  MoveL 8069 to (229.18, 36.07, 116.27) mm, rotated rx -180 ry 0 rz 180 deg; joints [-27.539, 54.39, -86.932, 31.738, 118.488, 16.437]
  MoveL 8070 to (229.18, 36.07, 116.27) mm, rotated rx -180 ry 0 rz 180 deg; joints [-27.539, 54.39, -86.932, 31.738, 118.488, 16.437]
  Call Extruder(197.85836)
  MoveL 8071 to (229.38, 36.12, 116.27) mm, rotated rx 180 ry 0 rz 180 deg; joints [-27.499, 54.413, -86.932, 31.688, 118.48, 16.403]
  MoveL 8072 to (229.38, 36.12, 116.27) mm, rotated rx 180 ry 0 rz 180 deg; joints [-27.499, 54.413, -86.932, 31.688, 118.48, 16.403]
  Call Extruder(197.97344)
  MoveL 8073 to (229.59, 36.16, 116.27) mm, rotated rx -180 ry 0 rz 180 deg; joints [-27.458, 54.436, -86.932, 31.638, 118.472, 16.368]
  MoveL 8074 to (229.59, 36.16, 116.27) mm, rotated rx -180 ry 0 rz 180 deg; joints [-27.458, 54.436, -86.932, 31.638, 118.472, 16.368]
  Call Extruder(198.09430)
  MoveL 8075 to (229.8, 36.21, 116.27) mm, rotated rx -180 ry 0 rz -180 deg; joints [-27.422, 54.459, -86.932, 31.591, 118.461, 16.335]
  MoveL 8076 to (229.8, 36.21, 116.27) mm, rotated rx -180 ry 0 rz -180 deg; joints [-27.422, 54.459, -86.932, 31.591, 118.461, 16.335]
  Call Extruder(198.22115)
  MoveL 8077 to (230.02, 36.28, 116.27) mm, rotated rx -180 ry 0 rz 180 deg; joints [-27.39, 54.485, -86.931, 31.549, 118.448, 16.303]
  MoveL 8078 to (230.02, 36.28, 116.27) mm, rotated rx -180 ry 0 rz 180 deg; joints [-27.39, 54.485, -86.931, 31.549, 118.448, 16.303]
  Call Extruder(198.33995)
  MoveL 8079 to (230.22, 36.34, 116.27) mm, rotated rx -180 ry 0 rz 180 deg; joints [-27.361, 54.508, -86.931, 31.51, 118.436, 16.274]
  MoveL 8080 to (230.22, 36.34, 116.27) mm, rotated rx -180 ry 0 rz 180 deg; joints [-27.361, 54.508, -86.931, 31.51, 118.436, 16.274]
  Call Extruder(198.45066)
  MoveL 8081 to (230.41, 36.4, 116.27) mm, rotated rx -180 ry 0 rz 180 deg; joints [-27.336, 54.53, -86.931, 31.477, 118.424, 16.248]
  MoveL 8082 to (230.41, 36.4, 116.27) mm, rotated rx -180 ry 0 rz 180 deg; joints [-27.336, 54.53, -86.931, 31.477, 118.424, 16.248]
  Call Extruder(198.56179)
  MoveL 8083 to (230.6, 36.46, 116.27) mm, rotated rx -180 ry 0 rz 180 deg; joints [-27.311, 54.552, -86.93, 31.444, 118.412, 16.222]
  MoveL 8084 to (230.6, 36.46, 116.27) mm, rotated rx -180 ry 0 rz 180 deg; joints [-27.311, 54.552, -86.93, 31.444, 118.412, 16.222]
  Call Extruder(198.67341)
  MoveL 8085 to (230.79, 36.52, 116.27) mm, rotated rx -180 ry 0 rz 180 deg; joints [-27.288, 54.574, -86.93, 31.412, 118.4, 16.196]
  MoveL 8086 to (230.79, 36.52, 116.27) mm, rotated rx -180 ry 0 rz 180 deg; joints [-27.288, 54.574, -86.93, 31.412, 118.4, 16.196]
  Call Extruder(198.78553)
  MoveL 8087 to (230.98, 36.58, 116.27) mm, rotated rx 180 ry 0 rz 180 deg; joints [-27.265, 54.596, -86.93, 31.381, 118.387, 16.171]
  MoveL 8088 to (230.98, 36.58, 116.27) mm, rotated rx 180 ry 0 rz 180 deg; joints [-27.265, 54.596, -86.93, 31.381, 118.387, 16.171]
  Call Extruder(198.89810)
  MoveL 8089 to (231.17, 36.64, 116.27) mm, rotated rx 180 ry 0 rz 180 deg; joints [-27.242, 54.618, -86.929, 31.349, 118.374, 16.146]
  MoveL 8090 to (231.17, 36.64, 116.27) mm, rotated rx 180 ry 0 rz 180 deg; joints [-27.242, 54.618, -86.929, 31.349, 118.374, 16.146]
  Call Extruder(199.01111)
  MoveL 8091 to (231.35, 36.7, 116.27) mm, rotated rx 180 ry 0 rz 180 deg; joints [-27.219, 54.64, -86.929, 31.318, 118.362, 16.121]
  MoveL 8092 to (231.35, 36.7, 116.27) mm, rotated rx 180 ry 0 rz 180 deg; joints [-27.219, 54.64, -86.929, 31.318, 118.362, 16.121]
  Call Extruder(199.12456)
  MoveL 8093 to (231.54, 36.76, 116.27) mm, rotated rx 180 ry 0 rz 180 deg; joints [-27.197, 54.662, -86.928, 31.287, 118.349, 16.096]
  MoveL 8094 to (231.54, 36.76, 116.27) mm, rotated rx 180 ry 0 rz 180 deg; joints [-27.197, 54.662, -86.928, 31.287, 118.349, 16.096]
  Call Extruder(199.27220)
  MoveL 8095 to (231.78, 36.85, 116.27) mm, rotated rx -180 ry 0 rz -180 deg; joints [-27.176, 54.691, -86.928, 31.257, 118.329, 16.068]
  MoveL 8096 to (231.78, 36.85, 116.27) mm, rotated rx -180 ry 0 rz -180 deg; joints [-27.176, 54.691, -86.928, 31.257, 118.329, 16.068]
  Call Extruder(199.45454)
  MoveL 8097 to (232.07, 36.97, 116.27) mm, rotated rx -180 ry 0 rz 180 deg; joints [-27.158, 54.726, -86.927, 31.227, 118.304, 16.038]
  MoveL 8098 to (232.07, 36.97, 116.27) mm, rotated rx -180 ry 0 rz 180 deg; joints [-27.158, 54.726, -86.927, 31.227, 118.304, 16.038]
  Call Extruder(199.63764)
  MoveL 8099 to (232.37, 37.1, 116.27) mm, rotated rx 180 ry 0 rz 180 deg; joints [-27.139, 54.761, -86.926, 31.196, 118.278, 16.007]
  MoveL 8100 to (232.37, 37.1, 116.27) mm, rotated rx 180 ry 0 rz 180 deg; joints [-27.139, 54.761, -86.926, 31.196, 118.278, 16.007]
  Call Extruder(199.79534)
  MoveL 8101 to (232.62, 37.2, 116.27) mm, rotated rx 180 ry 0 rz 180 deg; joints [-27.127, 54.791, -86.926, 31.174, 118.255, 15.982]
  MoveL 8102 to (232.62, 37.2, 116.27) mm, rotated rx 180 ry 0 rz 180 deg; joints [-27.127, 54.791, -86.926, 31.174, 118.255, 15.982]
  Call Extruder(199.95364)
  MoveL 8103 to (232.87, 37.31, 116.27) mm, rotated rx -180 ry 0 rz -180 deg; joints [-27.114, 54.822, -86.925, 31.151, 118.232, 15.957]
  MoveL 8104 to (232.87, 37.31, 116.27) mm, rotated rx -180 ry 0 rz -180 deg; joints [-27.114, 54.822, -86.925, 31.151, 118.232, 15.957]
  Call Extruder(200.13566)
  MoveL 8105 to (233.14, 37.45, 116.27) mm, rotated rx -180 ry 0 rz 180 deg; joints [-27.114, 54.856, -86.924, 31.141, 118.202, 15.936]
  MoveL 8106 to (233.14, 37.45, 116.27) mm, rotated rx -180 ry 0 rz 180 deg; joints [-27.114, 54.856, -86.924, 31.141, 118.202, 15.936]
  Call Extruder(200.34222)
  MoveL 8107 to (233.45, 37.63, 116.27) mm, rotated rx 180 ry 0 rz 180 deg; joints [-27.126, 54.895, -86.923, 31.143, 118.164, 15.919]
  MoveL 8108 to (233.45, 37.63, 116.27) mm, rotated rx 180 ry 0 rz 180 deg; joints [-27.126, 54.895, -86.923, 31.143, 118.164, 15.919]
  Call Extruder(200.54955)
  MoveL 8109 to (233.75, 37.8, 116.27) mm, rotated rx -180 ry 0 rz 180 deg; joints [-27.138, 54.935, -86.922, 31.145, 118.126, 15.901]
  MoveL 8110 to (233.75, 37.8, 116.27) mm, rotated rx -180 ry 0 rz 180 deg; joints [-27.138, 54.935, -86.922, 31.145, 118.126, 15.901]
  Call Extruder(200.75767)
  MoveL 8111 to (234.05, 37.98, 116.27) mm, rotated rx 180 ry 0 rz -180 deg; joints [-27.15, 54.974, -86.921, 31.148, 118.089, 15.884]
  MoveL 8112 to (234.05, 37.98, 116.27) mm, rotated rx 180 ry 0 rz -180 deg; joints [-27.15, 54.974, -86.921, 31.148, 118.089, 15.884]
  Call Extruder(200.87539)
  MoveL 8113 to (234.23, 38.08, 116.27) mm, rotated rx 180 ry 0 rz 180 deg; joints [-27.157, 54.996, -86.921, 31.149, 118.067, 15.875]
  MoveL 8114 to (234.23, 38.08, 116.27) mm, rotated rx 180 ry 0 rz 180 deg; joints [-27.157, 54.996, -86.921, 31.149, 118.067, 15.875]
  Call Extruder(201.20821)
  MoveL 8115 to (234.68, 38.4, 116.27) mm, rotated rx -180 ry 0 rz 180 deg; joints [-27.216, 55.057, -86.919, 31.196, 117.997, 15.868]
  MoveL 8116 to (234.68, 38.4, 116.27) mm, rotated rx -180 ry 0 rz 180 deg; joints [-27.216, 55.057, -86.919, 31.196, 117.997, 15.868]
  Call Extruder(201.54222)
  MoveL 8117 to (235.13, 38.73, 116.27) mm, rotated rx -180 ry 0 rz 180 deg; joints [-27.274, 55.119, -86.917, 31.241, 117.927, 15.86]
  MoveL 8118 to (235.13, 38.73, 116.27) mm, rotated rx -180 ry 0 rz 180 deg; joints [-27.274, 55.119, -86.917, 31.241, 117.927, 15.86]
  Call Extruder(201.70980)
  MoveL 8119 to (235.35, 38.9, 116.27) mm, rotated rx -180 ry 0 rz 180 deg; joints [-27.302, 55.149, -86.916, 31.264, 117.892, 15.856]
  Call Extruder(202.53913)
  MoveL 8120 to (236.39, 39.81, 116.27) mm, rotated rx 180 ry 0 rz 180 deg; joints [-27.525, 55.298, -86.91, 31.463, 117.7, 15.878]
  Call Extruder(203.17020)
  MoveL 8121 to (237.09, 40.59, 116.27) mm, rotated rx -180 ry 0 rz -180 deg; joints [-27.771, 55.407, -86.906, 31.7, 117.536, 15.935]
  MoveL 8122 to (237.09, 40.59, 116.27) mm, rotated rx -180 ry 0 rz -180 deg; joints [-27.771, 55.407, -86.906, 31.7, 117.536, 15.935]
  Call Extruder(203.36780)
  MoveL 8123 to (237.3, 40.85, 116.27) mm, rotated rx 180 ry 0 rz 180 deg; joints [-27.851, 55.441, -86.905, 31.777, 117.484, 15.954]
  Call Extruder(203.70181)
  MoveL 8124 to (237.63, 41.3, 116.27) mm, rotated rx 180 ry 0 rz 180 deg; joints [-28.012, 55.496, -86.902, 31.935, 117.39, 16]
  MoveL 8125 to (237.63, 41.3, 116.27) mm, rotated rx 180 ry 0 rz 180 deg; joints [-28.012, 55.496, -86.902, 31.935, 117.39, 16]
  Call Extruder(204.03463)
  MoveL 8126 to (237.96, 41.75, 116.27) mm, rotated rx 180 ry 0 rz 180 deg; joints [-28.17, 55.551, -86.9, 32.09, 117.298, 16.044]
  MoveL 8127 to (237.96, 41.75, 116.27) mm, rotated rx 180 ry 0 rz 180 deg; joints [-28.17, 55.551, -86.9, 32.09, 117.298, 16.044]
  Call Extruder(204.21387)
  MoveL 8128 to (238.13, 41.99, 116.27) mm, rotated rx 180 ry 0 rz 180 deg; joints [-28.256, 55.581, -86.898, 32.174, 117.247, 16.068]
  MoveL 8129 to (238.13, 41.99, 116.27) mm, rotated rx 180 ry 0 rz 180 deg; joints [-28.256, 55.581, -86.898, 32.174, 117.247, 16.068]
  Call Extruder(204.42198)
  MoveL 8130 to (238.31, 42.3, 116.27) mm, rotated rx -180 ry 0 rz 180 deg; joints [-28.375, 55.614, -86.897, 32.293, 117.185, 16.106]
  MoveL 8131 to (238.31, 42.3, 116.27) mm, rotated rx -180 ry 0 rz 180 deg; joints [-28.375, 55.614, -86.897, 32.293, 117.185, 16.106]
  Call Extruder(204.62931)
  MoveL 8132 to (238.49, 42.6, 116.27) mm, rotated rx -180 ry 0 rz -180 deg; joints [-28.493, 55.647, -86.895, 32.412, 117.123, 16.143]
  MoveL 8133 to (238.49, 42.6, 116.27) mm, rotated rx -180 ry 0 rz -180 deg; joints [-28.493, 55.647, -86.895, 32.412, 117.123, 16.143]
  Call Extruder(204.83587)
  MoveL 8134 to (238.66, 42.91, 116.27) mm, rotated rx -180 ry 0 rz -180 deg; joints [-28.61, 55.68, -86.893, 32.528, 117.061, 16.18]
  MoveL 8135 to (238.66, 42.91, 116.27) mm, rotated rx -180 ry 0 rz -180 deg; joints [-28.61, 55.68, -86.893, 32.528, 117.061, 16.18]
  Call Extruder(205.04165)
  MoveL 8136 to (238.84, 43.21, 116.27) mm, rotated rx -180 ry 0 rz 180 deg; joints [-28.727, 55.713, -86.892, 32.645, 117, 16.216]
  MoveL 8137 to (238.84, 43.21, 116.27) mm, rotated rx -180 ry 0 rz 180 deg; joints [-28.727, 55.713, -86.892, 32.645, 117, 16.216]
  Call Extruder(205.19996)
  MoveL 8138 to (238.94, 43.46, 116.27) mm, rotated rx -180 ry 0 rz 180 deg; joints [-28.834, 55.737, -86.89, 32.753, 116.949, 16.253]
  MoveL 8139 to (238.94, 43.46, 116.27) mm, rotated rx -180 ry 0 rz 180 deg; joints [-28.834, 55.737, -86.89, 32.753, 116.949, 16.253]
  Call Extruder(205.35767)
  MoveL 8140 to (239.05, 43.71, 116.27) mm, rotated rx 180 ry 0 rz 180 deg; joints [-28.939, 55.76, -86.889, 32.86, 116.899, 16.29]
  MoveL 8141 to (239.05, 43.71, 116.27) mm, rotated rx 180 ry 0 rz 180 deg; joints [-28.939, 55.76, -86.889, 32.86, 116.899, 16.29]
  Call Extruder(205.52776)
  MoveL 8142 to (239.17, 43.98, 116.27) mm, rotated rx 180 ry 0 rz 180 deg; joints [-29.054, 55.785, -86.888, 32.976, 116.844, 16.329]
  MoveL 8143 to (239.17, 43.98, 116.27) mm, rotated rx 180 ry 0 rz 180 deg; joints [-29.054, 55.785, -86.888, 32.976, 116.844, 16.329]
  Call Extruder(205.71010)
  MoveL 8144 to (239.29, 44.27, 116.27) mm, rotated rx -180 ry 0 rz 180 deg; joints [-29.178, 55.813, -86.886, 33.101, 116.785, 16.372]
  MoveL 8145 to (239.29, 44.27, 116.27) mm, rotated rx -180 ry 0 rz 180 deg; joints [-29.178, 55.813, -86.886, 33.101, 116.785, 16.372]
  Call Extruder(205.89168)
  MoveL 8146 to (239.41, 44.56, 116.27) mm, rotated rx 180 ry 0 rz -180 deg; joints [-29.301, 55.84, -86.885, 33.226, 116.726, 16.414]
  MoveL 8147 to (239.41, 44.56, 116.27) mm, rotated rx 180 ry 0 rz -180 deg; joints [-29.301, 55.84, -86.885, 33.226, 116.726, 16.414]
  Call Extruder(206.00513)
  MoveL 8148 to (239.47, 44.75, 116.27) mm, rotated rx -180 ry 0 rz 180 deg; joints [-29.385, 55.856, -86.884, 33.311, 116.688, 16.444]
  MoveL 8149 to (239.47, 44.75, 116.27) mm, rotated rx -180 ry 0 rz 180 deg; joints [-29.385, 55.856, -86.884, 33.311, 116.688, 16.444]
  Call Extruder(206.11815)
  MoveL 8150 to (239.53, 44.94, 116.27) mm, rotated rx 180 ry 0 rz -180 deg; joints [-29.47, 55.872, -86.883, 33.397, 116.65, 16.475]
  MoveL 8151 to (239.53, 44.94, 116.27) mm, rotated rx 180 ry 0 rz -180 deg; joints [-29.47, 55.872, -86.883, 33.397, 116.65, 16.475]
  Call Extruder(206.23072)
  MoveL 8152 to (239.59, 45.13, 116.27) mm, rotated rx -180 ry 0 rz 180 deg; joints [-29.553, 55.888, -86.882, 33.482, 116.612, 16.504]
  MoveL 8153 to (239.59, 45.13, 116.27) mm, rotated rx -180 ry 0 rz 180 deg; joints [-29.553, 55.888, -86.882, 33.482, 116.612, 16.504]
  Call Extruder(206.34284)
  MoveL 8154 to (239.65, 45.32, 116.27) mm, rotated rx 180 ry 0 rz -180 deg; joints [-29.637, 55.904, -86.881, 33.568, 116.574, 16.534]
  MoveL 8155 to (239.65, 45.32, 116.27) mm, rotated rx 180 ry 0 rz -180 deg; joints [-29.637, 55.904, -86.881, 33.568, 116.574, 16.534]
  Call Extruder(206.45452)
  MoveL 8156 to (239.71, 45.51, 116.27) mm, rotated rx 180 ry 0 rz 180 deg; joints [-29.72, 55.92, -86.88, 33.652, 116.537, 16.563]
  MoveL 8157 to (239.71, 45.51, 116.27) mm, rotated rx 180 ry 0 rz 180 deg; joints [-29.72, 55.92, -86.88, 33.652, 116.537, 16.563]
  Call Extruder(206.58559)
  MoveL 8158 to (239.78, 45.73, 116.27) mm, rotated rx -180 ry 0 rz 180 deg; joints [-29.821, 55.939, -86.879, 33.754, 116.492, 16.599]
  MoveL 8159 to (239.78, 45.73, 116.27) mm, rotated rx -180 ry 0 rz 180 deg; joints [-29.821, 55.939, -86.879, 33.754, 116.492, 16.599]
  Call Extruder(206.71610)
  MoveL 8160 to (239.85, 45.95, 116.27) mm, rotated rx 180 ry 0 rz -180 deg; joints [-29.921, 55.957, -86.878, 33.856, 116.447, 16.635]
  MoveL 8161 to (239.85, 45.95, 116.27) mm, rotated rx 180 ry 0 rz -180 deg; joints [-29.921, 55.957, -86.878, 33.856, 116.447, 16.635]
  Call Extruder(206.84604)
  MoveL 8162 to (239.92, 46.18, 116.27) mm, rotated rx -180 ry 0 rz 180 deg; joints [-30.02, 55.976, -86.877, 33.956, 116.402, 16.669]
  MoveL 8163 to (239.92, 46.18, 116.27) mm, rotated rx -180 ry 0 rz 180 deg; joints [-30.02, 55.976, -86.877, 33.956, 116.402, 16.669]
  Call Extruder(206.97542)
  MoveL 8164 to (239.98, 46.4, 116.27) mm, rotated rx -180 ry 0 rz 180 deg; joints [-30.119, 55.995, -86.876, 34.056, 116.357, 16.704]
  MoveL 8165 to (239.98, 46.4, 116.27) mm, rotated rx -180 ry 0 rz 180 deg; joints [-30.119, 55.995, -86.876, 34.056, 116.357, 16.704]
  Call Extruder(207.09738)
  MoveL 8166 to (240.04, 46.61, 116.27) mm, rotated rx -180 ry 0 rz 180 deg; joints [-30.216, 56.012, -86.875, 34.155, 116.314, 16.739]
  MoveL 8167 to (240.04, 46.61, 116.27) mm, rotated rx -180 ry 0 rz 180 deg; joints [-30.216, 56.012, -86.875, 34.155, 116.314, 16.739]
  Call Extruder(207.21220)
  MoveL 8168 to (240.08, 46.82, 116.27) mm, rotated rx -180 ry 0 rz 180 deg; joints [-30.311, 56.027, -86.874, 34.252, 116.273, 16.774]
  MoveL 8169 to (240.08, 46.82, 116.27) mm, rotated rx -180 ry 0 rz 180 deg; joints [-30.311, 56.027, -86.874, 34.252, 116.273, 16.774]
  Call Extruder(207.32658)
  MoveL 8170 to (240.13, 47.02, 116.27) mm, rotated rx -180 ry 0 rz 180 deg; joints [-30.406, 56.042, -86.873, 34.349, 116.232, 16.808]
  MoveL 8171 to (240.13, 47.02, 116.27) mm, rotated rx -180 ry 0 rz 180 deg; joints [-30.406, 56.042, -86.873, 34.349, 116.232, 16.808]
  Call Extruder(207.44050)
  MoveL 8172 to (240.17, 47.23, 116.27) mm, rotated rx 180 ry 0 rz 180 deg; joints [-30.5, 56.058, -86.872, 34.445, 116.191, 16.842]
  MoveL 8173 to (240.17, 47.23, 116.27) mm, rotated rx 180 ry 0 rz 180 deg; joints [-30.5, 56.058, -86.872, 34.445, 116.191, 16.842]
  Call Extruder(207.55397)
  MoveL 8174 to (240.22, 47.43, 116.27) mm, rotated rx 180 ry 0 rz 180 deg; joints [-30.595, 56.073, -86.871, 34.541, 116.15, 16.876]
  MoveL 8175 to (240.22, 47.43, 116.27) mm, rotated rx 180 ry 0 rz 180 deg; joints [-30.595, 56.073, -86.871, 34.541, 116.15, 16.876]
  Call Extruder(207.69125)
  MoveL 8176 to (240.27, 47.68, 116.27) mm, rotated rx 180 ry 0 rz 180 deg; joints [-30.711, 56.092, -86.869, 34.659, 116.1, 16.918]
  MoveL 8177 to (240.27, 47.68, 116.27) mm, rotated rx 180 ry 0 rz 180 deg; joints [-30.711, 56.092, -86.869, 34.659, 116.1, 16.918]
  Call Extruder(207.82792)
  MoveL 8178 to (240.32, 47.93, 116.27) mm, rotated rx -180 ry 0 rz 180 deg; joints [-30.827, 56.111, -86.868, 34.777, 116.05, 16.96]
  MoveL 8179 to (240.32, 47.93, 116.27) mm, rotated rx -180 ry 0 rz 180 deg; joints [-30.827, 56.111, -86.868, 34.777, 116.05, 16.96]
  Call Extruder(207.96399)
  MoveL 8180 to (240.37, 48.18, 116.27) mm, rotated rx -180 ry 0 rz 180 deg; joints [-30.942, 56.129, -86.867, 34.894, 116, 17.001]
  MoveL 8181 to (240.37, 48.18, 116.27) mm, rotated rx -180 ry 0 rz 180 deg; joints [-30.942, 56.129, -86.867, 34.894, 116, 17.001]
  Call Extruder(208.09944)
  MoveL 8182 to (240.42, 48.43, 116.27) mm, rotated rx -180 ry 0 rz 180 deg; joints [-31.057, 56.148, -86.866, 35.011, 115.95, 17.042]
  MoveL 8183 to (240.42, 48.43, 116.27) mm, rotated rx -180 ry 0 rz 180 deg; joints [-31.057, 56.148, -86.866, 35.011, 115.95, 17.042]
  Call Extruder(208.23428)
  MoveL 8184 to (240.47, 48.68, 116.27) mm, rotated rx 180 ry 0 rz 180 deg; joints [-31.171, 56.166, -86.865, 35.127, 115.901, 17.082]
  MoveL 8185 to (240.47, 48.68, 116.27) mm, rotated rx 180 ry 0 rz 180 deg; joints [-31.171, 56.166, -86.865, 35.127, 115.901, 17.082]
  Call Extruder(208.36851)
  MoveL 8186 to (240.52, 48.93, 116.27) mm, rotated rx -180 ry 0 rz 180 deg; joints [-31.285, 56.185, -86.863, 35.242, 115.851, 17.122]
  MoveL 8187 to (240.52, 48.93, 116.27) mm, rotated rx -180 ry 0 rz 180 deg; joints [-31.285, 56.185, -86.863, 35.242, 115.851, 17.122]
  Call Extruder(208.50213)
  MoveL 8188 to (240.57, 49.17, 116.27) mm, rotated rx -180 ry 0 rz 180 deg; joints [-31.398, 56.204, -86.862, 35.357, 115.801, 17.162]
  MoveL 8189 to (240.57, 49.17, 116.27) mm, rotated rx -180 ry 0 rz 180 deg; joints [-31.398, 56.204, -86.862, 35.357, 115.801, 17.162]
  Call Extruder(208.66424)
  MoveL 8190 to (240.61, 49.48, 116.27) mm, rotated rx -180 ry 0 rz 180 deg; joints [-31.541, 56.226, -86.861, 35.502, 115.74, 17.213]
  MoveL 8191 to (240.61, 49.48, 116.27) mm, rotated rx -180 ry 0 rz 180 deg; joints [-31.541, 56.226, -86.861, 35.502, 115.74, 17.213]
  Call Extruder(208.82562)
  MoveL 8192 to (240.66, 49.79, 116.27) mm, rotated rx -180 ry 0 rz 180 deg; joints [-31.684, 56.248, -86.859, 35.647, 115.678, 17.263]
  MoveL 8193 to (240.66, 49.79, 116.27) mm, rotated rx -180 ry 0 rz 180 deg; joints [-31.684, 56.248, -86.859, 35.647, 115.678, 17.263]
  Call Extruder(208.98628)
  MoveL 8194 to (240.71, 50.09, 116.27) mm, rotated rx -180 ry 0 rz 180 deg; joints [-31.825, 56.27, -86.857, 35.79, 115.617, 17.313]
  MoveL 8195 to (240.71, 50.09, 116.27) mm, rotated rx -180 ry 0 rz 180 deg; joints [-31.825, 56.27, -86.857, 35.79, 115.617, 17.313]
  Call Extruder(209.14620)
  MoveL 8196 to (240.76, 50.4, 116.27) mm, rotated rx -180 ry 0 rz 180 deg; joints [-31.966, 56.292, -86.856, 35.932, 115.556, 17.362]
  MoveL 8197 to (240.76, 50.4, 116.27) mm, rotated rx -180 ry 0 rz 180 deg; joints [-31.966, 56.292, -86.856, 35.932, 115.556, 17.362]
  Call Extruder(209.30540)
  MoveL 8198 to (240.81, 50.7, 116.27) mm, rotated rx -180 ry 0 rz 180 deg; joints [-32.106, 56.314, -86.854, 36.074, 115.495, 17.41]
  MoveL 8199 to (240.81, 50.7, 116.27) mm, rotated rx -180 ry 0 rz 180 deg; joints [-32.106, 56.314, -86.854, 36.074, 115.495, 17.41]
  Call Extruder(209.46387)
  MoveL 8200 to (240.86, 51.01, 116.27) mm, rotated rx -180 ry 0 rz 180 deg; joints [-32.246, 56.336, -86.853, 36.215, 115.434, 17.458]
  MoveL 8201 to (240.86, 51.01, 116.27) mm, rotated rx -180 ry 0 rz 180 deg; joints [-32.246, 56.336, -86.853, 36.215, 115.434, 17.458]
  Call Extruder(209.66274)
  MoveL 8202 to (240.9, 51.4, 116.27) mm, rotated rx 180 ry 0 rz 180 deg; joints [-32.427, 56.363, -86.851, 36.398, 115.357, 17.522]
  MoveL 8203 to (240.9, 51.4, 116.27) mm, rotated rx 180 ry 0 rz 180 deg; joints [-32.427, 56.363, -86.851, 36.398, 115.357, 17.522]
  Call Extruder(209.86075)
  MoveL 8204 to (240.95, 51.78, 116.27) mm, rotated rx 180 ry 0 rz 180 deg; joints [-32.608, 56.389, -86.849, 36.581, 115.279, 17.584]
  MoveL 8205 to (240.95, 51.78, 116.27) mm, rotated rx 180 ry 0 rz 180 deg; joints [-32.608, 56.389, -86.849, 36.581, 115.279, 17.584]
  Call Extruder(210.05789)
  MoveL 8206 to (240.99, 52.17, 116.27) mm, rotated rx -180 ry 0 rz 180 deg; joints [-32.787, 56.416, -86.847, 36.761, 115.202, 17.646]
  MoveL 8207 to (240.99, 52.17, 116.27) mm, rotated rx -180 ry 0 rz 180 deg; joints [-32.787, 56.416, -86.847, 36.761, 115.202, 17.646]
  Call Extruder(210.25416)
  MoveL 8208 to (241.04, 52.56, 116.27) mm, rotated rx -180 ry 0 rz 180 deg; joints [-32.966, 56.443, -86.845, 36.941, 115.124, 17.706]
  MoveL 8209 to (241.04, 52.56, 116.27) mm, rotated rx -180 ry 0 rz 180 deg; joints [-32.966, 56.443, -86.845, 36.941, 115.124, 17.706]
  Call Extruder(210.49987)
  MoveL 8210 to (241.09, 53.05, 116.27) mm, rotated rx 180 ry 0 rz 180 deg; joints [-33.193, 56.476, -86.842, 37.17, 115.026, 17.784]
  MoveL 8211 to (241.09, 53.05, 116.27) mm, rotated rx 180 ry 0 rz 180 deg; joints [-33.193, 56.476, -86.842, 37.17, 115.026, 17.784]
  Call Extruder(210.79465)
  MoveL 8212 to (241.13, 53.64, 116.27) mm, rotated rx -180 ry 0 rz 180 deg; joints [-33.469, 56.516, -86.839, 37.448, 114.908, 17.878]
  MoveL 8213 to (241.13, 53.64, 116.27) mm, rotated rx -180 ry 0 rz 180 deg; joints [-33.469, 56.516, -86.839, 37.448, 114.908, 17.878]
  Call Extruder(211.08809)
  MoveL 8214 to (241.18, 54.23, 116.27) mm, rotated rx 180 ry 0 rz 180 deg; joints [-33.742, 56.555, -86.836, 37.723, 114.79, 17.97]
  MoveL 8215 to (241.18, 54.23, 116.27) mm, rotated rx 180 ry 0 rz 180 deg; joints [-33.742, 56.555, -86.836, 37.723, 114.79, 17.97]
  Call Extruder(211.52144)
  MoveL 8216 to (241.22, 55.1, 116.27) mm, rotated rx 180 ry 0 rz 180 deg; joints [-34.152, 56.612, -86.831, 38.135, 114.615, 18.107]
  MoveL 8217 to (241.22, 55.1, 116.27) mm, rotated rx 180 ry 0 rz 180 deg; joints [-34.152, 56.612, -86.831, 38.135, 114.615, 18.107]
  Call Extruder(212.09360)
  MoveL 8218 to (241.27, 56.26, 116.27) mm, rotated rx 180 ry 0 rz 180 deg; joints [-34.696, 56.687, -86.825, 38.679, 114.381, 18.287]
  MoveL 8219 to (241.27, 56.26, 116.27) mm, rotated rx 180 ry 0 rz 180 deg; joints [-34.696, 56.687, -86.825, 38.679, 114.381, 18.287]
  Call Extruder(212.52130)
  MoveL 8220 to (241.29, 57.14, 116.27) mm, rotated rx 180 ry 0 rz 180 deg; joints [-35.104, 56.742, -86.82, 39.087, 114.206, 18.421]
  Call Extruder(254.51494)
  MoveL 8221 to (241.29, 142.86, 116.27) mm, rotated rx 180 ry 0 rz 180 deg; joints [-60.361, 63.196, -85.406, 62.221, 100.774, 19.538]
  MoveL 8222 to (241.29, 142.86, 116.27) mm, rotated rx 180 ry 0 rz 180 deg; joints [-60.361, 63.196, -85.406, 62.221, 100.774, 19.538]
  Call Extruder(255.23038)
  MoveL 8223 to (241.25, 144.32, 116.27) mm, rotated rx -180 ry 0 rz 180 deg; joints [-60.621, 63.308, -85.363, 62.445, 100.615, 19.445]
  MoveL 8224 to (241.25, 144.32, 116.27) mm, rotated rx -180 ry 0 rz 180 deg; joints [-60.621, 63.308, -85.363, 62.445, 100.615, 19.445]
  Call Extruder(255.80512)
  MoveL 8225 to (241.2, 145.48, 116.27) mm, rotated rx 180 ry 0 rz 180 deg; joints [-60.831, 63.397, -85.328, 62.626, 100.488, 19.37]
  MoveL 8226 to (241.2, 145.48, 116.27) mm, rotated rx 180 ry 0 rz 180 deg; joints [-60.831, 63.397, -85.328, 62.626, 100.488, 19.37]
  Call Extruder(256.09856)
  MoveL 8227 to (241.16, 146.07, 116.27) mm, rotated rx 180 ry 0 rz 180 deg; joints [-60.944, 63.441, -85.311, 62.724, 100.423, 19.334]
  MoveL 8228 to (241.16, 146.07, 116.27) mm, rotated rx 180 ry 0 rz 180 deg; joints [-60.944, 63.441, -85.311, 62.724, 100.423, 19.334]
  Call Extruder(256.39333)
  MoveL 8229 to (241.11, 146.66, 116.27) mm, rotated rx 180 ry 0 rz 180 deg; joints [-61.055, 63.485, -85.294, 62.821, 100.358, 19.298]
  MoveL 8230 to (241.11, 146.66, 116.27) mm, rotated rx 180 ry 0 rz 180 deg; joints [-61.055, 63.485, -85.294, 62.821, 100.358, 19.298]
  Call Extruder(256.68944)
  MoveL 8231 to (241.06, 147.25, 116.27) mm, rotated rx 180 ry 0 rz 180 deg; joints [-61.167, 63.529, -85.276, 62.918, 100.293, 19.261]
  MoveL 8232 to (241.06, 147.25, 116.27) mm, rotated rx 180 ry 0 rz 180 deg; joints [-61.167, 63.529, -85.276, 62.918, 100.293, 19.261]
  Call Extruder(256.88571)
  MoveL 8233 to (241.02, 147.63, 116.27) mm, rotated rx -180 ry 0 rz -180 deg; joints [-61.244, 63.558, -85.265, 62.985, 100.25, 19.239]
  MoveL 8234 to (241.02, 147.63, 116.27) mm, rotated rx -180 ry 0 rz -180 deg; joints [-61.244, 63.558, -85.265, 62.985, 100.25, 19.239]
  Call Extruder(257.08285)
  MoveL 8235 to (240.97, 148.02, 116.27) mm, rotated rx 180 ry 0 rz 180 deg; joints [-61.321, 63.586, -85.253, 63.053, 100.206, 19.216]
  MoveL 8236 to (240.97, 148.02, 116.27) mm, rotated rx 180 ry 0 rz 180 deg; joints [-61.321, 63.586, -85.253, 63.053, 100.206, 19.216]
  Call Extruder(257.28085)
  MoveL 8237 to (240.93, 148.41, 116.27) mm, rotated rx -180 ry 0 rz 180 deg; joints [-61.397, 63.614, -85.242, 63.12, 100.163, 19.193]
  MoveL 8238 to (240.93, 148.41, 116.27) mm, rotated rx -180 ry 0 rz 180 deg; joints [-61.397, 63.614, -85.242, 63.12, 100.163, 19.193]
  Call Extruder(257.47973)
  MoveL 8239 to (240.88, 148.8, 116.27) mm, rotated rx 180 ry 0 rz 180 deg; joints [-61.474, 63.643, -85.23, 63.187, 100.12, 19.17]
  MoveL 8240 to (240.88, 148.8, 116.27) mm, rotated rx 180 ry 0 rz 180 deg; joints [-61.474, 63.643, -85.23, 63.187, 100.12, 19.17]
  Call Extruder(257.65881)
  MoveL 8241 to (240.83, 149.14, 116.27) mm, rotated rx 180 ry 0 rz 180 deg; joints [-61.544, 63.668, -85.22, 63.248, 100.081, 19.15]
  MoveL 8242 to (240.83, 149.14, 116.27) mm, rotated rx 180 ry 0 rz 180 deg; joints [-61.544, 63.668, -85.22, 63.248, 100.081, 19.15]
  Call Extruder(257.81801)
  MoveL 8243 to (240.78, 149.45, 116.27) mm, rotated rx -180 ry 0 rz -180 deg; joints [-61.607, 63.69, -85.211, 63.305, 100.046, 19.132]
  MoveL 8244 to (240.78, 149.45, 116.27) mm, rotated rx -180 ry 0 rz -180 deg; joints [-61.607, 63.69, -85.211, 63.305, 100.046, 19.132]
  Call Extruder(257.97794)
  MoveL 8245 to (240.74, 149.76, 116.27) mm, rotated rx 180 ry 0 rz 180 deg; joints [-61.67, 63.711, -85.202, 63.36, 100.012, 19.115]
  MoveL 8246 to (240.74, 149.76, 116.27) mm, rotated rx 180 ry 0 rz 180 deg; joints [-61.67, 63.711, -85.202, 63.36, 100.012, 19.115]
  Call Extruder(258.13859)
  MoveL 8247 to (240.69, 150.06, 116.27) mm, rotated rx -180 ry 0 rz 180 deg; joints [-61.734, 63.733, -85.194, 63.416, 99.977, 19.098]
  MoveL 8248 to (240.69, 150.06, 116.27) mm, rotated rx -180 ry 0 rz 180 deg; joints [-61.734, 63.733, -85.194, 63.416, 99.977, 19.098]
  Call Extruder(258.29997)
  MoveL 8249 to (240.64, 150.37, 116.27) mm, rotated rx 180 ry 0 rz 180 deg; joints [-61.796, 63.755, -85.185, 63.472, 99.943, 19.08]
  MoveL 8250 to (240.64, 150.37, 116.27) mm, rotated rx 180 ry 0 rz 180 deg; joints [-61.796, 63.755, -85.185, 63.472, 99.943, 19.08]
  Call Extruder(258.46208)
  MoveL 8251 to (240.59, 150.67, 116.27) mm, rotated rx 180 ry 0 rz -180 deg; joints [-61.859, 63.777, -85.176, 63.527, 99.909, 19.063]
  MoveL 8252 to (240.59, 150.67, 116.27) mm, rotated rx 180 ry 0 rz -180 deg; joints [-61.859, 63.777, -85.176, 63.527, 99.909, 19.063]
  Call Extruder(258.61028)
  MoveL 8253 to (240.54, 150.95, 116.27) mm, rotated rx -180 ry 0 rz -180 deg; joints [-61.918, 63.796, -85.167, 63.579, 99.877, 19.047]
  MoveL 8254 to (240.54, 150.95, 116.27) mm, rotated rx -180 ry 0 rz -180 deg; joints [-61.918, 63.796, -85.167, 63.579, 99.877, 19.047]
  Call Extruder(258.74452)
  MoveL 8255 to (240.49, 151.2, 116.27) mm, rotated rx -180 ry 0 rz 180 deg; joints [-61.971, 63.814, -85.16, 63.626, 99.849, 19.033]
  MoveL 8256 to (240.49, 151.2, 116.27) mm, rotated rx -180 ry 0 rz 180 deg; joints [-61.971, 63.814, -85.16, 63.626, 99.849, 19.033]
  Call Extruder(258.87936)
  MoveL 8257 to (240.44, 151.45, 116.27) mm, rotated rx -180 ry 0 rz 180 deg; joints [-62.025, 63.831, -85.153, 63.674, 99.821, 19.02]
  MoveL 8258 to (240.44, 151.45, 116.27) mm, rotated rx -180 ry 0 rz 180 deg; joints [-62.025, 63.831, -85.153, 63.674, 99.821, 19.02]
  Call Extruder(259.01481)
  MoveL 8259 to (240.39, 151.7, 116.27) mm, rotated rx -180 ry 0 rz 180 deg; joints [-62.079, 63.848, -85.146, 63.722, 99.792, 19.006]
  MoveL 8260 to (240.39, 151.7, 116.27) mm, rotated rx -180 ry 0 rz 180 deg; joints [-62.079, 63.848, -85.146, 63.722, 99.792, 19.006]
  Call Extruder(259.15087)
  MoveL 8261 to (240.34, 151.95, 116.27) mm, rotated rx -180 ry 0 rz 180 deg; joints [-62.132, 63.866, -85.138, 63.769, 99.764, 18.993]
  MoveL 8262 to (240.34, 151.95, 116.27) mm, rotated rx -180 ry 0 rz 180 deg; joints [-62.132, 63.866, -85.138, 63.769, 99.764, 18.993]
  Call Extruder(259.28754)
  MoveL 8263 to (240.29, 152.2, 116.27) mm, rotated rx -180 ry 0 rz 180 deg; joints [-62.186, 63.883, -85.131, 63.817, 99.736, 18.979]
  MoveL 8264 to (240.29, 152.2, 116.27) mm, rotated rx -180 ry 0 rz 180 deg; joints [-62.186, 63.883, -85.131, 63.817, 99.736, 18.979]
  Call Extruder(259.42483)
  MoveL 8265 to (240.24, 152.45, 116.27) mm, rotated rx 180 ry 0 rz -180 deg; joints [-62.239, 63.901, -85.124, 63.864, 99.707, 18.965]
  MoveL 8266 to (240.24, 152.45, 116.27) mm, rotated rx 180 ry 0 rz -180 deg; joints [-62.239, 63.901, -85.124, 63.864, 99.707, 18.965]
  Call Extruder(259.55049)
  MoveL 8267 to (240.2, 152.67, 116.27) mm, rotated rx 180 ry 0 rz 180 deg; joints [-62.288, 63.916, -85.117, 63.907, 99.682, 18.952]
  MoveL 8268 to (240.2, 152.67, 116.27) mm, rotated rx 180 ry 0 rz 180 deg; joints [-62.288, 63.916, -85.117, 63.907, 99.682, 18.952]
  Call Extruder(259.66441)
  MoveL 8269 to (240.15, 152.88, 116.27) mm, rotated rx -180 ry 0 rz 180 deg; joints [-62.333, 63.93, -85.111, 63.947, 99.658, 18.941]
  MoveL 8270 to (240.15, 152.88, 116.27) mm, rotated rx -180 ry 0 rz 180 deg; joints [-62.333, 63.93, -85.111, 63.947, 99.658, 18.941]
  Call Extruder(259.77879)
  MoveL 8271 to (240.11, 153.08, 116.27) mm, rotated rx -180 ry 0 rz 180 deg; joints [-62.377, 63.944, -85.105, 63.987, 99.635, 18.93]
  MoveL 8272 to (240.11, 153.08, 116.27) mm, rotated rx -180 ry 0 rz 180 deg; joints [-62.377, 63.944, -85.105, 63.987, 99.635, 18.93]
  Call Extruder(259.89362)
  MoveL 8273 to (240.06, 153.28, 116.27) mm, rotated rx 180 ry 0 rz -180 deg; joints [-62.421, 63.958, -85.099, 64.027, 99.612, 18.919]
  MoveL 8274 to (240.06, 153.28, 116.27) mm, rotated rx 180 ry 0 rz -180 deg; joints [-62.421, 63.958, -85.099, 64.027, 99.612, 18.919]
  Call Extruder(260.00890)
  MoveL 8275 to (240.02, 153.49, 116.27) mm, rotated rx -180 ry 0 rz -180 deg; joints [-62.466, 63.973, -85.093, 64.066, 99.589, 18.908]
  MoveL 8276 to (240.02, 153.49, 116.27) mm, rotated rx -180 ry 0 rz -180 deg; joints [-62.466, 63.973, -85.093, 64.066, 99.589, 18.908]
  Call Extruder(260.13828)
  MoveL 8277 to (239.95, 153.71, 116.27) mm, rotated rx 180 ry 0 rz -180 deg; joints [-62.52, 63.987, -85.087, 64.115, 99.562, 18.897]
  MoveL 8278 to (239.95, 153.71, 116.27) mm, rotated rx 180 ry 0 rz -180 deg; joints [-62.52, 63.987, -85.087, 64.115, 99.562, 18.897]
  Call Extruder(260.26822)
  MoveL 8279 to (239.88, 153.94, 116.27) mm, rotated rx -180 ry 0 rz 180 deg; joints [-62.574, 64.002, -85.081, 64.163, 99.535, 18.887]
  MoveL 8280 to (239.88, 153.94, 116.27) mm, rotated rx -180 ry 0 rz 180 deg; joints [-62.574, 64.002, -85.081, 64.163, 99.535, 18.887]
  Call Extruder(260.39873)
  MoveL 8281 to (239.81, 154.16, 116.27) mm, rotated rx -180 ry 0 rz 180 deg; joints [-62.627, 64.017, -85.074, 64.212, 99.509, 18.876]
  MoveL 8282 to (239.81, 154.16, 116.27) mm, rotated rx -180 ry 0 rz 180 deg; joints [-62.627, 64.017, -85.074, 64.212, 99.509, 18.876]
  Call Extruder(260.52980)
  MoveL 8283 to (239.75, 154.38, 116.27) mm, rotated rx 180 ry 0 rz -180 deg; joints [-62.681, 64.031, -85.068, 64.26, 99.482, 18.866]
  MoveL 8284 to (239.75, 154.38, 116.27) mm, rotated rx 180 ry 0 rz -180 deg; joints [-62.681, 64.031, -85.068, 64.26, 99.482, 18.866]
  Call Extruder(260.65144)
  MoveL 8285 to (239.68, 154.59, 116.27) mm, rotated rx -180 ry 0 rz 180 deg; joints [-62.731, 64.045, -85.062, 64.305, 99.458, 18.856]
  MoveL 8286 to (239.68, 154.59, 116.27) mm, rotated rx -180 ry 0 rz 180 deg; joints [-62.731, 64.045, -85.062, 64.305, 99.458, 18.856]
  Call Extruder(260.76357)
  MoveL 8287 to (239.62, 154.78, 116.27) mm, rotated rx 180 ry 0 rz 180 deg; joints [-62.778, 64.057, -85.057, 64.347, 99.435, 18.847]
  MoveL 8288 to (239.62, 154.78, 116.27) mm, rotated rx 180 ry 0 rz 180 deg; joints [-62.778, 64.057, -85.057, 64.347, 99.435, 18.847]
  Call Extruder(260.87613)
  MoveL 8289 to (239.56, 154.97, 116.27) mm, rotated rx -180 ry 0 rz 180 deg; joints [-62.824, 64.069, -85.052, 64.389, 99.413, 18.839]
  MoveL 8290 to (239.56, 154.97, 116.27) mm, rotated rx -180 ry 0 rz 180 deg; joints [-62.824, 64.069, -85.052, 64.389, 99.413, 18.839]
  Call Extruder(260.98915)
  MoveL 8291 to (239.5, 155.15, 116.27) mm, rotated rx 180 ry 0 rz -180 deg; joints [-62.87, 64.081, -85.046, 64.43, 99.39, 18.83]
  MoveL 8292 to (239.5, 155.15, 116.27) mm, rotated rx 180 ry 0 rz -180 deg; joints [-62.87, 64.081, -85.046, 64.43, 99.39, 18.83]
  Call Extruder(261.10260)
  MoveL 8293 to (239.44, 155.34, 116.27) mm, rotated rx -180 ry 0 rz 180 deg; joints [-62.916, 64.094, -85.041, 64.472, 99.368, 18.821]
  MoveL 8294 to (239.44, 155.34, 116.27) mm, rotated rx -180 ry 0 rz 180 deg; joints [-62.916, 64.094, -85.041, 64.472, 99.368, 18.821]
  Call Extruder(261.25025)
  MoveL 8295 to (239.35, 155.58, 116.27) mm, rotated rx 180 ry 0 rz 180 deg; joints [-62.979, 64.109, -85.035, 64.529, 99.338, 18.811]
  MoveL 8296 to (239.35, 155.58, 116.27) mm, rotated rx 180 ry 0 rz 180 deg; joints [-62.979, 64.109, -85.035, 64.529, 99.338, 18.811]
  Call Extruder(261.43258)
  MoveL 8297 to (239.23, 155.88, 116.27) mm, rotated rx -180 ry 0 rz 180 deg; joints [-63.058, 64.126, -85.027, 64.601, 99.302, 18.8]
  MoveL 8298 to (239.23, 155.88, 116.27) mm, rotated rx -180 ry 0 rz 180 deg; joints [-63.058, 64.126, -85.027, 64.601, 99.302, 18.8]
  Call Extruder(261.61568)
  MoveL 8299 to (239.11, 156.17, 116.27) mm, rotated rx 180 ry 0 rz 180 deg; joints [-63.136, 64.144, -85.019, 64.672, 99.266, 18.788]
  MoveL 8300 to (239.11, 156.17, 116.27) mm, rotated rx 180 ry 0 rz 180 deg; joints [-63.136, 64.144, -85.019, 64.672, 99.266, 18.788]
  Call Extruder(261.77338)
  MoveL 8301 to (239, 156.42, 116.27) mm, rotated rx 180 ry 0 rz 180 deg; joints [-63.204, 64.16, -85.012, 64.734, 99.234, 18.779]
  MoveL 8302 to (239, 156.42, 116.27) mm, rotated rx 180 ry 0 rz 180 deg; joints [-63.204, 64.16, -85.012, 64.734, 99.234, 18.779]
  Call Extruder(261.93170)
  MoveL 8303 to (238.89, 156.66, 116.27) mm, rotated rx -180 ry 0 rz 180 deg; joints [-63.272, 64.175, -85.006, 64.796, 99.203, 18.769]
  MoveL 8304 to (238.89, 156.66, 116.27) mm, rotated rx -180 ry 0 rz 180 deg; joints [-63.272, 64.175, -85.006, 64.796, 99.203, 18.769]
  Call Extruder(262.11373)
  MoveL 8305 to (238.75, 156.94, 116.27) mm, rotated rx 180 ry 0 rz 180 deg; joints [-63.354, 64.191, -84.999, 64.871, 99.167, 18.761]
  MoveL 8306 to (238.75, 156.94, 116.27) mm, rotated rx 180 ry 0 rz 180 deg; joints [-63.354, 64.191, -84.999, 64.871, 99.167, 18.761]
  Call Extruder(262.32029)
  MoveL 8307 to (238.57, 157.25, 116.27) mm, rotated rx -180 ry 0 rz -180 deg; joints [-63.449, 64.208, -84.991, 64.959, 99.126, 18.753]
  MoveL 8308 to (238.57, 157.25, 116.27) mm, rotated rx -180 ry 0 rz -180 deg; joints [-63.449, 64.208, -84.991, 64.959, 99.126, 18.753]
  Call Extruder(262.52763)
  MoveL 8309 to (238.4, 157.55, 116.27) mm, rotated rx 180 ry 0 rz 180 deg; joints [-63.544, 64.224, -84.984, 65.047, 99.085, 18.745]
  MoveL 8310 to (238.4, 157.55, 116.27) mm, rotated rx 180 ry 0 rz 180 deg; joints [-63.544, 64.224, -84.984, 65.047, 99.085, 18.745]
  Call Extruder(262.73575)
  MoveL 8311 to (238.22, 157.85, 116.27) mm, rotated rx 180 ry 0 rz -180 deg; joints [-63.64, 64.241, -84.976, 65.135, 99.044, 18.737]
  MoveL 8312 to (238.22, 157.85, 116.27) mm, rotated rx 180 ry 0 rz -180 deg; joints [-63.64, 64.241, -84.976, 65.135, 99.044, 18.737]
  Call Extruder(262.85347)
  MoveL 8313 to (238.12, 158.03, 116.27) mm, rotated rx -180 ry 0 rz 180 deg; joints [-63.693, 64.251, -84.972, 65.184, 99.021, 18.732]
  MoveL 8314 to (238.12, 158.03, 116.27) mm, rotated rx -180 ry 0 rz 180 deg; joints [-63.693, 64.251, -84.972, 65.184, 99.021, 18.732]
  Call Extruder(263.18629)
  MoveL 8315 to (237.8, 158.48, 116.27) mm, rotated rx -180 ry 0 rz 180 deg; joints [-63.854, 64.273, -84.962, 65.334, 98.956, 18.727]
  MoveL 8316 to (237.8, 158.48, 116.27) mm, rotated rx -180 ry 0 rz 180 deg; joints [-63.854, 64.273, -84.962, 65.334, 98.956, 18.727]
  Call Extruder(263.52029)
  MoveL 8317 to (237.47, 158.93, 116.27) mm, rotated rx -180 ry 0 rz 180 deg; joints [-64.014, 64.296, -84.952, 65.482, 98.891, 18.72]
  MoveL 8318 to (237.47, 158.93, 116.27) mm, rotated rx -180 ry 0 rz 180 deg; joints [-64.014, 64.296, -84.952, 65.482, 98.891, 18.72]
  Call Extruder(263.68786)
  MoveL 8319 to (237.3, 159.15, 116.27) mm, rotated rx 180 ry 0 rz 180 deg; joints [-64.094, 64.307, -84.947, 65.556, 98.859, 18.717]
  Call Extruder(264.51719)
  MoveL 8320 to (236.39, 160.19, 116.27) mm, rotated rx -180 ry 0 rz 180 deg; joints [-64.505, 64.354, -84.926, 65.941, 98.699, 18.714]
  Call Extruder(265.14825)
  MoveL 8321 to (235.6, 160.89, 116.27) mm, rotated rx 180 ry 0 rz 180 deg; joints [-64.83, 64.379, -84.914, 66.248, 98.58, 18.727]
  MoveL 8322 to (235.6, 160.89, 116.27) mm, rotated rx 180 ry 0 rz 180 deg; joints [-64.83, 64.379, -84.914, 66.248, 98.58, 18.727]
  Call Extruder(265.34587)
  MoveL 8323 to (235.35, 161.1, 116.27) mm, rotated rx -180 ry 0 rz -180 deg; joints [-64.933, 64.387, -84.911, 66.344, 98.542, 18.732]
  Call Extruder(265.67988)
  MoveL 8324 to (234.9, 161.43, 116.27) mm, rotated rx -180 ry 0 rz 180 deg; joints [-65.109, 64.396, -84.907, 66.511, 98.48, 18.744]
  MoveL 8325 to (234.9, 161.43, 116.27) mm, rotated rx -180 ry 0 rz 180 deg; joints [-65.109, 64.396, -84.907, 66.511, 98.48, 18.744]
  Call Extruder(266.01272)
  MoveL 8326 to (234.45, 161.76, 116.27) mm, rotated rx 180 ry 0 rz 180 deg; joints [-65.285, 64.406, -84.902, 66.678, 98.418, 18.756]
  MoveL 8327 to (234.45, 161.76, 116.27) mm, rotated rx 180 ry 0 rz 180 deg; joints [-65.285, 64.406, -84.902, 66.678, 98.418, 18.756]
  Call Extruder(266.19191)
  MoveL 8328 to (234.21, 161.93, 116.27) mm, rotated rx -180 ry 0 rz 180 deg; joints [-65.381, 64.411, -84.9, 66.768, 98.385, 18.763]
  MoveL 8329 to (234.21, 161.93, 116.27) mm, rotated rx -180 ry 0 rz 180 deg; joints [-65.381, 64.411, -84.9, 66.768, 98.385, 18.763]
  Call Extruder(266.40003)
  MoveL 8330 to (233.9, 162.11, 116.27) mm, rotated rx 180 ry 0 rz -180 deg; joints [-65.493, 64.413, -84.899, 66.875, 98.347, 18.775]
  MoveL 8331 to (233.9, 162.11, 116.27) mm, rotated rx 180 ry 0 rz -180 deg; joints [-65.493, 64.413, -84.899, 66.875, 98.347, 18.775]
  Call Extruder(266.60737)
  MoveL 8332 to (233.6, 162.29, 116.27) mm, rotated rx 180 ry 0 rz -180 deg; joints [-65.605, 64.416, -84.897, 66.982, 98.309, 18.786]
  MoveL 8333 to (233.6, 162.29, 116.27) mm, rotated rx 180 ry 0 rz -180 deg; joints [-65.605, 64.416, -84.897, 66.982, 98.309, 18.786]
  Call Extruder(266.81392)
  MoveL 8334 to (233.29, 162.46, 116.27) mm, rotated rx -180 ry 0 rz 180 deg; joints [-65.718, 64.419, -84.896, 67.089, 98.271, 18.798]
  MoveL 8335 to (233.29, 162.46, 116.27) mm, rotated rx -180 ry 0 rz 180 deg; joints [-65.718, 64.419, -84.896, 67.089, 98.271, 18.798]
  Call Extruder(267.01970)
  MoveL 8336 to (232.99, 162.64, 116.27) mm, rotated rx 180 ry 0 rz -180 deg; joints [-65.83, 64.422, -84.895, 67.196, 98.233, 18.809]
  MoveL 8337 to (232.99, 162.64, 116.27) mm, rotated rx 180 ry 0 rz -180 deg; joints [-65.83, 64.422, -84.895, 67.196, 98.233, 18.809]
  Call Extruder(267.17798)
  MoveL 8338 to (232.74, 162.74, 116.27) mm, rotated rx -180 ry 0 rz 180 deg; joints [-65.917, 64.422, -84.895, 67.279, 98.205, 18.821]
  MoveL 8339 to (232.74, 162.74, 116.27) mm, rotated rx -180 ry 0 rz 180 deg; joints [-65.917, 64.422, -84.895, 67.279, 98.205, 18.821]
  Call Extruder(267.33565)
  MoveL 8340 to (232.49, 162.85, 116.27) mm, rotated rx -180 ry 0 rz -180 deg; joints [-66.004, 64.422, -84.895, 67.363, 98.177, 18.834]
  MoveL 8341 to (232.49, 162.85, 116.27) mm, rotated rx -180 ry 0 rz -180 deg; joints [-66.004, 64.422, -84.895, 67.363, 98.177, 18.834]
  Call Extruder(267.50574)
  MoveL 8342 to (232.22, 162.97, 116.27) mm, rotated rx 180 ry 0 rz 180 deg; joints [-66.099, 64.421, -84.895, 67.453, 98.147, 18.847]
  MoveL 8343 to (232.22, 162.97, 116.27) mm, rotated rx 180 ry 0 rz 180 deg; joints [-66.099, 64.421, -84.895, 67.453, 98.147, 18.847]
  Call Extruder(267.68811)
  MoveL 8344 to (231.93, 163.09, 116.27) mm, rotated rx -180 ry 0 rz 180 deg; joints [-66.2, 64.421, -84.895, 67.55, 98.115, 18.862]
  MoveL 8345 to (231.93, 163.09, 116.27) mm, rotated rx -180 ry 0 rz 180 deg; joints [-66.2, 64.421, -84.895, 67.55, 98.115, 18.862]
  Call Extruder(267.86971)
  MoveL 8346 to (231.64, 163.21, 116.27) mm, rotated rx -180 ry 0 rz 180 deg; joints [-66.302, 64.42, -84.896, 67.647, 98.082, 18.876]
  MoveL 8347 to (231.64, 163.21, 116.27) mm, rotated rx -180 ry 0 rz 180 deg; joints [-66.302, 64.42, -84.896, 67.647, 98.082, 18.876]
  Call Extruder(267.98315)
  MoveL 8348 to (231.45, 163.27, 116.27) mm, rotated rx -180 ry 0 rz -180 deg; joints [-66.365, 64.418, -84.896, 67.708, 98.063, 18.887]
  MoveL 8349 to (231.45, 163.27, 116.27) mm, rotated rx -180 ry 0 rz -180 deg; joints [-66.365, 64.418, -84.896, 67.708, 98.063, 18.887]
  Call Extruder(268.09615)
  MoveL 8350 to (231.26, 163.33, 116.27) mm, rotated rx 180 ry 0 rz -180 deg; joints [-66.428, 64.417, -84.897, 67.769, 98.043, 18.898]
  MoveL 8351 to (231.26, 163.33, 116.27) mm, rotated rx 180 ry 0 rz -180 deg; joints [-66.428, 64.417, -84.897, 67.769, 98.043, 18.898]
  Call Extruder(268.20871)
  MoveL 8352 to (231.07, 163.39, 116.27) mm, rotated rx -180 ry 0 rz 180 deg; joints [-66.492, 64.415, -84.898, 67.83, 98.023, 18.909]
  MoveL 8353 to (231.07, 163.39, 116.27) mm, rotated rx -180 ry 0 rz 180 deg; joints [-66.492, 64.415, -84.898, 67.83, 98.023, 18.909]
  Call Extruder(268.32082)
  MoveL 8354 to (230.88, 163.45, 116.27) mm, rotated rx 180 ry 0 rz 180 deg; joints [-66.555, 64.413, -84.899, 67.891, 98.004, 18.919]
  MoveL 8355 to (230.88, 163.45, 116.27) mm, rotated rx 180 ry 0 rz 180 deg; joints [-66.555, 64.413, -84.899, 67.891, 98.004, 18.919]
  Call Extruder(268.43249)
  MoveL 8356 to (230.69, 163.51, 116.27) mm, rotated rx -180 ry 0 rz -180 deg; joints [-66.619, 64.412, -84.899, 67.952, 97.984, 18.93]
  MoveL 8357 to (230.69, 163.51, 116.27) mm, rotated rx -180 ry 0 rz -180 deg; joints [-66.619, 64.412, -84.899, 67.952, 97.984, 18.93]
  Call Extruder(268.56358)
  MoveL 8358 to (230.47, 163.58, 116.27) mm, rotated rx -180 ry 0 rz 180 deg; joints [-66.694, 64.409, -84.9, 68.024, 97.961, 18.943]
  MoveL 8359 to (230.47, 163.58, 116.27) mm, rotated rx -180 ry 0 rz 180 deg; joints [-66.694, 64.409, -84.9, 68.024, 97.961, 18.943]
  Call Extruder(268.69411)
  MoveL 8360 to (230.25, 163.65, 116.27) mm, rotated rx 180 ry 0 rz 180 deg; joints [-66.768, 64.407, -84.902, 68.096, 97.938, 18.956]
  MoveL 8361 to (230.25, 163.65, 116.27) mm, rotated rx 180 ry 0 rz 180 deg; joints [-66.768, 64.407, -84.902, 68.096, 97.938, 18.956]
  Call Extruder(268.82408)
  MoveL 8362 to (230.02, 163.72, 116.27) mm, rotated rx 180 ry 0 rz 180 deg; joints [-66.843, 64.405, -84.903, 68.167, 97.915, 18.969]
  MoveL 8363 to (230.02, 163.72, 116.27) mm, rotated rx 180 ry 0 rz 180 deg; joints [-66.843, 64.405, -84.903, 68.167, 97.915, 18.969]
  Call Extruder(268.95347)
  MoveL 8364 to (229.8, 163.78, 116.27) mm, rotated rx -180 ry 0 rz -180 deg; joints [-66.918, 64.403, -84.904, 68.239, 97.892, 18.982]
  MoveL 8365 to (229.8, 163.78, 116.27) mm, rotated rx -180 ry 0 rz -180 deg; joints [-66.918, 64.403, -84.904, 68.239, 97.892, 18.982]
  Call Extruder(269.07545)
  MoveL 8366 to (229.59, 163.84, 116.27) mm, rotated rx 180 ry 0 rz 180 deg; joints [-66.988, 64.4, -84.905, 68.307, 97.871, 18.995]
  MoveL 8367 to (229.59, 163.84, 116.27) mm, rotated rx 180 ry 0 rz 180 deg; joints [-66.988, 64.4, -84.905, 68.307, 97.871, 18.995]
  Call Extruder(269.19030)
  MoveL 8368 to (229.38, 163.88, 116.27) mm, rotated rx -180 ry 0 rz -180 deg; joints [-67.054, 64.397, -84.906, 68.37, 97.851, 19.008]
  MoveL 8369 to (229.38, 163.88, 116.27) mm, rotated rx -180 ry 0 rz -180 deg; joints [-67.054, 64.397, -84.906, 68.37, 97.851, 19.008]
  Call Extruder(269.30469)
  MoveL 8370 to (229.18, 163.93, 116.27) mm, rotated rx 180 ry 0 rz 180 deg; joints [-67.12, 64.393, -84.908, 68.434, 97.831, 19.021]
  MoveL 8371 to (229.18, 163.93, 116.27) mm, rotated rx 180 ry 0 rz 180 deg; joints [-67.12, 64.393, -84.908, 68.434, 97.831, 19.021]
  Call Extruder(269.41863)
  MoveL 8372 to (228.97, 163.97, 116.27) mm, rotated rx -180 ry 0 rz 180 deg; joints [-67.187, 64.39, -84.909, 68.498, 97.811, 19.034]
  MoveL 8373 to (228.97, 163.97, 116.27) mm, rotated rx -180 ry 0 rz 180 deg; joints [-67.187, 64.39, -84.909, 68.498, 97.811, 19.034]
  Call Extruder(269.53212)
  MoveL 8374 to (228.77, 164.02, 116.27) mm, rotated rx -180 ry 0 rz 180 deg; joints [-67.253, 64.387, -84.911, 68.562, 97.791, 19.047]
  MoveL 8375 to (228.77, 164.02, 116.27) mm, rotated rx -180 ry 0 rz 180 deg; joints [-67.253, 64.387, -84.911, 68.562, 97.791, 19.047]
  Call Extruder(269.66941)
  MoveL 8376 to (228.52, 164.07, 116.27) mm, rotated rx 180 ry 0 rz 180 deg; joints [-67.333, 64.382, -84.913, 68.639, 97.767, 19.063]
  MoveL 8377 to (228.52, 164.07, 116.27) mm, rotated rx 180 ry 0 rz 180 deg; joints [-67.333, 64.382, -84.913, 68.639, 97.767, 19.063]
  Call Extruder(269.80608)
  MoveL 8378 to (228.27, 164.12, 116.27) mm, rotated rx -180 ry 0 rz -180 deg; joints [-67.413, 64.378, -84.915, 68.716, 97.744, 19.08]
  MoveL 8379 to (228.27, 164.12, 116.27) mm, rotated rx -180 ry 0 rz -180 deg; joints [-67.413, 64.378, -84.915, 68.716, 97.744, 19.08]
  Call Extruder(269.94214)
  MoveL 8380 to (228.02, 164.17, 116.27) mm, rotated rx -180 ry 0 rz -180 deg; joints [-67.494, 64.374, -84.917, 68.794, 97.72, 19.096]
  MoveL 8381 to (228.02, 164.17, 116.27) mm, rotated rx -180 ry 0 rz -180 deg; joints [-67.494, 64.374, -84.917, 68.794, 97.72, 19.096]
  Call Extruder(270.07759)
  MoveL 8382 to (227.77, 164.22, 116.27) mm, rotated rx 180 ry 0 rz -180 deg; joints [-67.574, 64.369, -84.919, 68.871, 97.696, 19.112]
  MoveL 8383 to (227.77, 164.22, 116.27) mm, rotated rx 180 ry 0 rz -180 deg; joints [-67.574, 64.369, -84.919, 68.871, 97.696, 19.112]
  Call Extruder(270.21244)
  MoveL 8384 to (227.52, 164.27, 116.27) mm, rotated rx -180 ry 0 rz 180 deg; joints [-67.654, 64.365, -84.921, 68.949, 97.671, 19.128]
  MoveL 8385 to (227.52, 164.27, 116.27) mm, rotated rx -180 ry 0 rz 180 deg; joints [-67.654, 64.365, -84.921, 68.949, 97.671, 19.128]
  Call Extruder(270.34667)
  MoveL 8386 to (227.28, 164.32, 116.27) mm, rotated rx -180 ry 0 rz 180 deg; joints [-67.735, 64.361, -84.922, 69.026, 97.647, 19.144]
  MoveL 8387 to (227.28, 164.32, 116.27) mm, rotated rx -180 ry 0 rz 180 deg; joints [-67.735, 64.361, -84.922, 69.026, 97.647, 19.144]
  Call Extruder(270.48029)
  MoveL 8388 to (227.02, 164.36, 116.27) mm, rotated rx -180 ry 0 rz 180 deg; joints [-67.815, 64.357, -84.924, 69.104, 97.623, 19.16]
  MoveL 8389 to (227.02, 164.36, 116.27) mm, rotated rx -180 ry 0 rz 180 deg; joints [-67.815, 64.357, -84.924, 69.104, 97.623, 19.16]
  Call Extruder(270.64240)
  MoveL 8390 to (226.72, 164.41, 116.27) mm, rotated rx -180 ry 0 rz -180 deg; joints [-67.912, 64.351, -84.927, 69.197, 97.594, 19.18]
  MoveL 8391 to (226.72, 164.41, 116.27) mm, rotated rx -180 ry 0 rz -180 deg; joints [-67.912, 64.351, -84.927, 69.197, 97.594, 19.18]
  Call Extruder(270.80377)
  MoveL 8392 to (226.41, 164.46, 116.27) mm, rotated rx 180 ry 0 rz 180 deg; joints [-68.01, 64.345, -84.93, 69.291, 97.565, 19.201]
  MoveL 8393 to (226.41, 164.46, 116.27) mm, rotated rx 180 ry 0 rz 180 deg; joints [-68.01, 64.345, -84.93, 69.291, 97.565, 19.201]
  Call Extruder(270.96442)
  MoveL 8394 to (226.11, 164.51, 116.27) mm, rotated rx -180 ry 0 rz -180 deg; joints [-68.107, 64.339, -84.933, 69.385, 97.536, 19.221]
  MoveL 8395 to (226.11, 164.51, 116.27) mm, rotated rx -180 ry 0 rz -180 deg; joints [-68.107, 64.339, -84.933, 69.385, 97.536, 19.221]
  Call Extruder(271.12435)
  MoveL 8396 to (225.8, 164.56, 116.27) mm, rotated rx -180 ry 0 rz 180 deg; joints [-68.205, 64.333, -84.935, 69.479, 97.507, 19.242]
  MoveL 8397 to (225.8, 164.56, 116.27) mm, rotated rx -180 ry 0 rz 180 deg; joints [-68.205, 64.333, -84.935, 69.479, 97.507, 19.242]
  Call Extruder(271.28354)
  MoveL 8398 to (225.5, 164.61, 116.27) mm, rotated rx -180 ry 0 rz 180 deg; joints [-68.303, 64.327, -84.938, 69.573, 97.478, 19.262]
  MoveL 8399 to (225.5, 164.61, 116.27) mm, rotated rx -180 ry 0 rz 180 deg; joints [-68.303, 64.327, -84.938, 69.573, 97.478, 19.262]
  Call Extruder(271.44201)
  MoveL 8400 to (225.19, 164.66, 116.27) mm, rotated rx -180 ry 0 rz -180 deg; joints [-68.4, 64.321, -84.941, 69.667, 97.449, 19.282]
  MoveL 8401 to (225.19, 164.66, 116.27) mm, rotated rx -180 ry 0 rz -180 deg; joints [-68.4, 64.321, -84.941, 69.667, 97.449, 19.282]
  Call Extruder(271.64088)
  MoveL 8402 to (224.8, 164.7, 116.27) mm, rotated rx -180 ry 0 rz 180 deg; joints [-68.522, 64.312, -84.944, 69.785, 97.413, 19.309]
  MoveL 8403 to (224.8, 164.7, 116.27) mm, rotated rx -180 ry 0 rz 180 deg; joints [-68.522, 64.312, -84.944, 69.785, 97.413, 19.309]
  Call Extruder(271.83889)
  MoveL 8404 to (224.42, 164.75, 116.27) mm, rotated rx -180 ry 0 rz 180 deg; joints [-68.645, 64.304, -84.948, 69.903, 97.376, 19.336]
  MoveL 8405 to (224.42, 164.75, 116.27) mm, rotated rx -180 ry 0 rz 180 deg; joints [-68.645, 64.304, -84.948, 69.903, 97.376, 19.336]
  Call Extruder(272.03603)
  MoveL 8406 to (224.03, 164.79, 116.27) mm, rotated rx -180 ry 0 rz 180 deg; joints [-68.767, 64.295, -84.952, 70.021, 97.34, 19.362]
  MoveL 8407 to (224.03, 164.79, 116.27) mm, rotated rx -180 ry 0 rz 180 deg; joints [-68.767, 64.295, -84.952, 70.021, 97.34, 19.362]
  Call Extruder(272.23230)
  MoveL 8408 to (223.64, 164.84, 116.27) mm, rotated rx 180 ry 0 rz 180 deg; joints [-68.89, 64.287, -84.956, 70.139, 97.304, 19.388]
  MoveL 8409 to (223.64, 164.84, 116.27) mm, rotated rx 180 ry 0 rz 180 deg; joints [-68.89, 64.287, -84.956, 70.139, 97.304, 19.388]
  Call Extruder(272.47797)
  MoveL 8410 to (223.15, 164.89, 116.27) mm, rotated rx -180 ry 0 rz -180 deg; joints [-69.043, 64.276, -84.961, 70.286, 97.258, 19.423]
  MoveL 8411 to (223.15, 164.89, 116.27) mm, rotated rx -180 ry 0 rz -180 deg; joints [-69.043, 64.276, -84.961, 70.286, 97.258, 19.423]
  Call Extruder(272.77266)
  MoveL 8412 to (222.56, 164.93, 116.27) mm, rotated rx -180 ry 0 rz 180 deg; joints [-69.227, 64.261, -84.967, 70.464, 97.204, 19.465]
  MoveL 8413 to (222.56, 164.93, 116.27) mm, rotated rx -180 ry 0 rz 180 deg; joints [-69.227, 64.261, -84.967, 70.464, 97.204, 19.465]
  Call Extruder(273.06601)
  MoveL 8414 to (221.97, 164.98, 116.27) mm, rotated rx 180 ry 0 rz 180 deg; joints [-69.411, 64.247, -84.974, 70.642, 97.149, 19.506]
  MoveL 8415 to (221.97, 164.98, 116.27) mm, rotated rx 180 ry 0 rz 180 deg; joints [-69.411, 64.247, -84.974, 70.642, 97.149, 19.506]
  Call Extruder(273.49932)
  MoveL 8416 to (221.1, 165.02, 116.27) mm, rotated rx 180 ry 0 rz -180 deg; joints [-69.684, 64.224, -84.984, 70.904, 97.069, 19.569]
  MoveL 8417 to (221.1, 165.02, 116.27) mm, rotated rx 180 ry 0 rz -180 deg; joints [-69.684, 64.224, -84.984, 70.904, 97.069, 19.569]
  Call Extruder(274.07148)
  MoveL 8418 to (219.94, 165.07, 116.27) mm, rotated rx -180 ry 0 rz 180 deg; joints [-70.044, 64.193, -84.998, 71.252, 96.963, 19.654]
  MoveL 8419 to (219.94, 165.07, 116.27) mm, rotated rx -180 ry 0 rz 180 deg; joints [-70.044, 64.193, -84.998, 71.252, 96.963, 19.654]
  Call Extruder(274.49936)
  MoveL 8420 to (219.06, 165.09, 116.27) mm, rotated rx -180 ry 0 rz 180 deg; joints [-70.315, 64.168, -85.008, 71.512, 96.883, 19.718]
  Call Extruder(391.14801)
  MoveL 8421 to (-19.06, 165.09, 116.27) mm, rotated rx 180 ry 0 rz 180 deg; joints [-137.325, 69.391, -81.52, 136.68, 81.113, 8.288]
  MoveL 8422 to (-19.06, 165.09, 116.27) mm, rotated rx 180 ry 0 rz 180 deg; joints [-137.325, 69.391, -81.52, 136.68, 81.113, 8.288]
  Call Extruder(391.86364)
  MoveL 8423 to (-20.52, 165.05, 116.27) mm, rotated rx -180 ry 0 rz 180 deg; joints [-137.563, 69.459, -81.453, 136.933, 81.178, 8.158]
  MoveL 8424 to (-20.52, 165.05, 116.27) mm, rotated rx -180 ry 0 rz 180 deg; joints [-137.563, 69.459, -81.453, 136.933, 81.178, 8.158]
  Call Extruder(392.43838)
  MoveL 8425 to (-21.68, 165, 116.27) mm, rotated rx 180 ry 0 rz 180 deg; joints [-137.754, 69.513, -81.4, 137.136, 81.23, 8.055]
  MoveL 8426 to (-21.68, 165, 116.27) mm, rotated rx 180 ry 0 rz 180 deg; joints [-137.754, 69.513, -81.4, 137.136, 81.23, 8.055]
  Call Extruder(392.73174)
  MoveL 8427 to (-22.27, 164.95, 116.27) mm, rotated rx -180 ry 0 rz 180 deg; joints [-137.855, 69.539, -81.373, 137.242, 81.254, 8.003]
  MoveL 8428 to (-22.27, 164.95, 116.27) mm, rotated rx -180 ry 0 rz 180 deg; joints [-137.855, 69.539, -81.373, 137.242, 81.254, 8.003]
  Call Extruder(393.02643)
  MoveL 8429 to (-22.86, 164.91, 116.27) mm, rotated rx 180 ry 0 rz -180 deg; joints [-137.955, 69.566, -81.347, 137.347, 81.279, 7.952]
  MoveL 8430 to (-22.86, 164.91, 116.27) mm, rotated rx 180 ry 0 rz -180 deg; joints [-137.955, 69.566, -81.347, 137.347, 81.279, 7.952]
  Call Extruder(393.32246)
  MoveL 8431 to (-23.45, 164.86, 116.27) mm, rotated rx 180 ry 0 rz -180 deg; joints [-138.054, 69.592, -81.321, 137.453, 81.304, 7.901]
  MoveL 8432 to (-23.45, 164.86, 116.27) mm, rotated rx 180 ry 0 rz -180 deg; joints [-138.054, 69.592, -81.321, 137.453, 81.304, 7.901]
  Call Extruder(393.51873)
  MoveL 8433 to (-23.84, 164.82, 116.27) mm, rotated rx 180 ry 0 rz 180 deg; joints [-138.122, 69.609, -81.304, 137.524, 81.319, 7.867]
  MoveL 8434 to (-23.84, 164.82, 116.27) mm, rotated rx 180 ry 0 rz 180 deg; joints [-138.122, 69.609, -81.304, 137.524, 81.319, 7.867]
  Call Extruder(393.71587)
  MoveL 8435 to (-24.22, 164.77, 116.27) mm, rotated rx -180 ry 0 rz 180 deg; joints [-138.19, 69.625, -81.287, 137.596, 81.335, 7.834]
  MoveL 8436 to (-24.22, 164.77, 116.27) mm, rotated rx -180 ry 0 rz 180 deg; joints [-138.19, 69.625, -81.287, 137.596, 81.335, 7.834]
  Call Extruder(393.91388)
  MoveL 8437 to (-24.61, 164.72, 116.27) mm, rotated rx 180 ry 0 rz -180 deg; joints [-138.258, 69.642, -81.27, 137.667, 81.35, 7.801]
  MoveL 8438 to (-24.61, 164.72, 116.27) mm, rotated rx 180 ry 0 rz -180 deg; joints [-138.258, 69.642, -81.27, 137.667, 81.35, 7.801]
  Call Extruder(394.11275)
  MoveL 8439 to (-25, 164.68, 116.27) mm, rotated rx 180 ry 0 rz 180 deg; joints [-138.325, 69.659, -81.253, 137.738, 81.366, 7.768]
  MoveL 8440 to (-25, 164.68, 116.27) mm, rotated rx 180 ry 0 rz 180 deg; joints [-138.325, 69.659, -81.253, 137.738, 81.366, 7.768]
  Call Extruder(394.29183)
  MoveL 8441 to (-25.34, 164.63, 116.27) mm, rotated rx 180 ry 0 rz 180 deg; joints [-138.387, 69.673, -81.238, 137.803, 81.38, 7.739]
  MoveL 8442 to (-25.34, 164.63, 116.27) mm, rotated rx 180 ry 0 rz 180 deg; joints [-138.387, 69.673, -81.238, 137.803, 81.38, 7.739]
  Call Extruder(394.45103)
  MoveL 8443 to (-25.65, 164.58, 116.27) mm, rotated rx 180 ry 0 rz 180 deg; joints [-138.442, 69.686, -81.225, 137.861, 81.391, 7.713]
  MoveL 8444 to (-25.65, 164.58, 116.27) mm, rotated rx 180 ry 0 rz 180 deg; joints [-138.442, 69.686, -81.225, 137.861, 81.391, 7.713]
  Call Extruder(394.61095)
  MoveL 8445 to (-25.96, 164.53, 116.27) mm, rotated rx -180 ry 0 rz 180 deg; joints [-138.497, 69.698, -81.212, 137.919, 81.403, 7.688]
  MoveL 8446 to (-25.96, 164.53, 116.27) mm, rotated rx -180 ry 0 rz 180 deg; joints [-138.497, 69.698, -81.212, 137.919, 81.403, 7.688]
  Call Extruder(394.77161)
  MoveL 8447 to (-26.26, 164.49, 116.27) mm, rotated rx -180 ry 0 rz -180 deg; joints [-138.552, 69.711, -81.199, 137.976, 81.414, 7.662]
  MoveL 8448 to (-26.26, 164.49, 116.27) mm, rotated rx -180 ry 0 rz -180 deg; joints [-138.552, 69.711, -81.199, 137.976, 81.414, 7.662]
  Call Extruder(394.93299)
  MoveL 8449 to (-26.57, 164.44, 116.27) mm, rotated rx -180 ry 0 rz -180 deg; joints [-138.607, 69.724, -81.186, 138.034, 81.426, 7.637]
  MoveL 8450 to (-26.57, 164.44, 116.27) mm, rotated rx -180 ry 0 rz -180 deg; joints [-138.607, 69.724, -81.186, 138.034, 81.426, 7.637]
  Call Extruder(395.09509)
  MoveL 8451 to (-26.87, 164.39, 116.27) mm, rotated rx 180 ry 0 rz 180 deg; joints [-138.662, 69.736, -81.173, 138.092, 81.438, 7.611]
  MoveL 8452 to (-26.87, 164.39, 116.27) mm, rotated rx 180 ry 0 rz 180 deg; joints [-138.662, 69.736, -81.173, 138.092, 81.438, 7.611]
  Call Extruder(395.24330)
  MoveL 8453 to (-27.15, 164.34, 116.27) mm, rotated rx -180 ry 0 rz -180 deg; joints [-138.713, 69.748, -81.162, 138.145, 81.448, 7.588]
  MoveL 8454 to (-27.15, 164.34, 116.27) mm, rotated rx -180 ry 0 rz -180 deg; joints [-138.713, 69.748, -81.162, 138.145, 81.448, 7.588]
  Call Extruder(395.37753)
  MoveL 8455 to (-27.4, 164.29, 116.27) mm, rotated rx -180 ry 0 rz 180 deg; joints [-138.759, 69.757, -81.152, 138.193, 81.457, 7.568]
  MoveL 8456 to (-27.4, 164.29, 116.27) mm, rotated rx -180 ry 0 rz 180 deg; joints [-138.759, 69.757, -81.152, 138.193, 81.457, 7.568]
  Call Extruder(395.51237)
  MoveL 8457 to (-27.65, 164.24, 116.27) mm, rotated rx -180 ry 0 rz -180 deg; joints [-138.806, 69.767, -81.141, 138.242, 81.466, 7.547]
  MoveL 8458 to (-27.65, 164.24, 116.27) mm, rotated rx -180 ry 0 rz -180 deg; joints [-138.806, 69.767, -81.141, 138.242, 81.466, 7.547]
  Call Extruder(395.64782)
  MoveL 8459 to (-27.9, 164.19, 116.27) mm, rotated rx 180 ry 0 rz -180 deg; joints [-138.852, 69.777, -81.131, 138.29, 81.475, 7.527]
  MoveL 8460 to (-27.9, 164.19, 116.27) mm, rotated rx 180 ry 0 rz -180 deg; joints [-138.852, 69.777, -81.131, 138.29, 81.475, 7.527]
  Call Extruder(395.78388)
  MoveL 8461 to (-28.15, 164.14, 116.27) mm, rotated rx -180 ry 0 rz -180 deg; joints [-138.898, 69.787, -81.121, 138.338, 81.484, 7.506]
  MoveL 8462 to (-28.15, 164.14, 116.27) mm, rotated rx -180 ry 0 rz -180 deg; joints [-138.898, 69.787, -81.121, 138.338, 81.484, 7.506]
  Call Extruder(395.92056)
  MoveL 8463 to (-28.4, 164.09, 116.27) mm, rotated rx 180 ry 0 rz 180 deg; joints [-138.944, 69.797, -81.111, 138.387, 81.493, 7.486]
  MoveL 8464 to (-28.4, 164.09, 116.27) mm, rotated rx 180 ry 0 rz 180 deg; joints [-138.944, 69.797, -81.111, 138.387, 81.493, 7.486]
  Call Extruder(396.05784)
  MoveL 8465 to (-28.64, 164.04, 116.27) mm, rotated rx -180 ry 0 rz 180 deg; joints [-138.99, 69.807, -81.1, 138.435, 81.502, 7.466]
  MoveL 8466 to (-28.64, 164.04, 116.27) mm, rotated rx -180 ry 0 rz 180 deg; joints [-138.99, 69.807, -81.1, 138.435, 81.502, 7.466]
  Call Extruder(396.18351)
  MoveL 8467 to (-28.87, 164, 116.27) mm, rotated rx 180 ry 0 rz 180 deg; joints [-139.032, 69.816, -81.091, 138.479, 81.51, 7.447]
  MoveL 8468 to (-28.87, 164, 116.27) mm, rotated rx 180 ry 0 rz 180 deg; joints [-139.032, 69.816, -81.091, 138.479, 81.51, 7.447]
  Call Extruder(396.29745)
  MoveL 8469 to (-29.08, 163.95, 116.27) mm, rotated rx 180 ry 0 rz 180 deg; joints [-139.071, 69.824, -81.083, 138.519, 81.517, 7.431]
  MoveL 8470 to (-29.08, 163.95, 116.27) mm, rotated rx 180 ry 0 rz 180 deg; joints [-139.071, 69.824, -81.083, 138.519, 81.517, 7.431]
  Call Extruder(396.41184)
  MoveL 8471 to (-29.28, 163.91, 116.27) mm, rotated rx 180 ry 0 rz -180 deg; joints [-139.109, 69.832, -81.074, 138.559, 81.524, 7.414]
  MoveL 8472 to (-29.28, 163.91, 116.27) mm, rotated rx 180 ry 0 rz -180 deg; joints [-139.109, 69.832, -81.074, 138.559, 81.524, 7.414]
  Call Extruder(396.52669)
  MoveL 8473 to (-29.48, 163.86, 116.27) mm, rotated rx -180 ry 0 rz 180 deg; joints [-139.147, 69.839, -81.066, 138.599, 81.532, 7.398]
  MoveL 8474 to (-29.48, 163.86, 116.27) mm, rotated rx -180 ry 0 rz 180 deg; joints [-139.147, 69.839, -81.066, 138.599, 81.532, 7.398]
  Call Extruder(396.64199)
  MoveL 8475 to (-29.69, 163.82, 116.27) mm, rotated rx -180 ry 0 rz 180 deg; joints [-139.186, 69.847, -81.058, 138.639, 81.539, 7.381]
  MoveL 8476 to (-29.69, 163.82, 116.27) mm, rotated rx -180 ry 0 rz 180 deg; joints [-139.186, 69.847, -81.058, 138.639, 81.539, 7.381]
  Call Extruder(396.77138)
  MoveL 8477 to (-29.91, 163.75, 116.27) mm, rotated rx 180 ry 0 rz 180 deg; joints [-139.231, 69.855, -81.049, 138.686, 81.545, 7.364]
  MoveL 8478 to (-29.91, 163.75, 116.27) mm, rotated rx 180 ry 0 rz 180 deg; joints [-139.231, 69.855, -81.049, 138.686, 81.545, 7.364]
  Call Extruder(396.90134)
  MoveL 8479 to (-30.14, 163.68, 116.27) mm, rotated rx -180 ry 0 rz 180 deg; joints [-139.276, 69.863, -81.041, 138.733, 81.552, 7.346]
  MoveL 8480 to (-30.14, 163.68, 116.27) mm, rotated rx -180 ry 0 rz 180 deg; joints [-139.276, 69.863, -81.041, 138.733, 81.552, 7.346]
  Call Extruder(397.03187)
  MoveL 8481 to (-30.36, 163.61, 116.27) mm, rotated rx -180 ry 0 rz -180 deg; joints [-139.321, 69.871, -81.033, 138.779, 81.558, 7.329]
  MoveL 8482 to (-30.36, 163.61, 116.27) mm, rotated rx -180 ry 0 rz -180 deg; joints [-139.321, 69.871, -81.033, 138.779, 81.558, 7.329]
  Call Extruder(397.16296)
  MoveL 8483 to (-30.58, 163.55, 116.27) mm, rotated rx -180 ry 0 rz -180 deg; joints [-139.366, 69.879, -81.024, 138.826, 81.565, 7.311]
  MoveL 8484 to (-30.58, 163.55, 116.27) mm, rotated rx -180 ry 0 rz -180 deg; joints [-139.366, 69.879, -81.024, 138.826, 81.565, 7.311]
  Call Extruder(397.28461)
  MoveL 8485 to (-30.79, 163.48, 116.27) mm, rotated rx 180 ry 0 rz 180 deg; joints [-139.408, 69.886, -81.017, 138.869, 81.571, 7.295]
  MoveL 8486 to (-30.79, 163.48, 116.27) mm, rotated rx 180 ry 0 rz 180 deg; joints [-139.408, 69.886, -81.017, 138.869, 81.571, 7.295]
  Call Extruder(397.39672)
  MoveL 8487 to (-30.98, 163.42, 116.27) mm, rotated rx 180 ry 0 rz 180 deg; joints [-139.446, 69.893, -81.01, 138.909, 81.576, 7.28]
  MoveL 8488 to (-30.98, 163.42, 116.27) mm, rotated rx 180 ry 0 rz 180 deg; joints [-139.446, 69.893, -81.01, 138.909, 81.576, 7.28]
  Call Extruder(397.50928)
  MoveL 8489 to (-31.17, 163.36, 116.27) mm, rotated rx -180 ry 0 rz 180 deg; joints [-139.485, 69.899, -81.003, 138.949, 81.581, 7.266]
  MoveL 8490 to (-31.17, 163.36, 116.27) mm, rotated rx -180 ry 0 rz 180 deg; joints [-139.485, 69.899, -81.003, 138.949, 81.581, 7.266]
  Call Extruder(397.54120)
  MoveL 8491 to (-31.22, 163.34, 116.27) mm, rotated rx -180 ry 0 rz 180 deg; joints [-139.495, 69.901, -81.001, 138.96, 81.583, 7.262]
  Set speed (130.0 mm/s)
  MoveL 8492 to (-34.34, 162.18, 116.27) mm, rotated rx 180 ry 0 rz 180 deg; joints [-140.155, 70.004, -80.891, 139.642, 81.662, 7.026]
  MoveL 8493 to (-34.34, 162.18, 125.68) mm, rotated rx -180 ry 0 rz -180 deg; joints [-140.155, 71.36, -82.678, 139.6, 81.333, 7.308]
  MoveL 8494 to (-31.64, 163.21, 125.68) mm, rotated rx 180 ry 0 rz 180 deg; joints [-139.581, 71.27, -82.773, 139.006, 81.268, 7.516]
  Set speed (30.0 mm/s)
  MoveL 8495 to (-31.64, 163.21, 125.68) mm, rotated rx 180 ry 0 rz 180 deg; joints [-139.581, 71.27, -82.773, 139.006, 81.268, 7.516]
  Call Extruder(397.72317)
  MoveL 8496 to (-31.93, 163.09, 125.68) mm, rotated rx 180 ry 0 rz 180 deg; joints [-139.645, 71.28, -82.763, 139.072, 81.274, 7.494]
  MoveL 8497 to (-31.93, 163.09, 125.68) mm, rotated rx 180 ry 0 rz 180 deg; joints [-139.645, 71.28, -82.763, 139.072, 81.274, 7.494]
  Call Extruder(397.90591)
  MoveL 8498 to (-32.22, 162.97, 125.68) mm, rotated rx 180 ry 0 rz -180 deg; joints [-139.709, 71.289, -82.754, 139.138, 81.28, 7.472]
  MoveL 8499 to (-32.22, 162.97, 125.68) mm, rotated rx 180 ry 0 rz -180 deg; joints [-139.709, 71.289, -82.754, 139.138, 81.28, 7.472]
  Call Extruder(398.07632)
  MoveL 8500 to (-32.49, 162.85, 125.68) mm, rotated rx -180 ry 0 rz -180 deg; joints [-139.768, 71.297, -82.745, 139.2, 81.285, 7.451]
  MoveL 8501 to (-32.49, 162.85, 125.68) mm, rotated rx -180 ry 0 rz -180 deg; joints [-139.768, 71.297, -82.745, 139.2, 81.285, 7.451]
  Call Extruder(398.23430)
  MoveL 8502 to (-32.74, 162.74, 125.68) mm, rotated rx 180 ry 0 rz 180 deg; joints [-139.823, 71.305, -82.737, 139.257, 81.29, 7.432]
  MoveL 8503 to (-32.74, 162.74, 125.68) mm, rotated rx 180 ry 0 rz 180 deg; joints [-139.823, 71.305, -82.737, 139.257, 81.29, 7.432]
  Call Extruder(398.39287)
  MoveL 8504 to (-32.99, 162.64, 125.68) mm, rotated rx 180 ry 0 rz 180 deg; joints [-139.878, 71.313, -82.728, 139.313, 81.295, 7.413]
  MoveL 8505 to (-32.99, 162.64, 125.68) mm, rotated rx 180 ry 0 rz 180 deg; joints [-139.878, 71.313, -82.728, 139.313, 81.295, 7.413]
  Call Extruder(398.59904)
  MoveL 8506 to (-33.29, 162.46, 125.68) mm, rotated rx -180 ry 0 rz -180 deg; joints [-139.953, 71.321, -82.72, 139.39, 81.297, 7.392]
  MoveL 8507 to (-33.29, 162.46, 125.68) mm, rotated rx -180 ry 0 rz -180 deg; joints [-139.953, 71.321, -82.72, 139.39, 81.297, 7.392]
  Call Extruder(398.80598)
  MoveL 8508 to (-33.6, 162.29, 125.68) mm, rotated rx -180 ry 0 rz -180 deg; joints [-140.028, 71.328, -82.712, 139.467, 81.3, 7.37]
  MoveL 8509 to (-33.6, 162.29, 125.68) mm, rotated rx -180 ry 0 rz -180 deg; joints [-140.028, 71.328, -82.712, 139.467, 81.3, 7.37]
  Call Extruder(399.01371)
  MoveL 8510 to (-33.9, 162.11, 125.68) mm, rotated rx -180 ry 0 rz 180 deg; joints [-140.103, 71.336, -82.704, 139.543, 81.302, 7.348]
  MoveL 8511 to (-33.9, 162.11, 125.68) mm, rotated rx -180 ry 0 rz 180 deg; joints [-140.103, 71.336, -82.704, 139.543, 81.302, 7.348]
  Call Extruder(399.22221)
  MoveL 8512 to (-34.21, 161.93, 125.68) mm, rotated rx 180 ry 0 rz 180 deg; joints [-140.178, 71.344, -82.696, 139.62, 81.305, 7.327]
  MoveL 8513 to (-34.21, 161.93, 125.68) mm, rotated rx 180 ry 0 rz 180 deg; joints [-140.178, 71.344, -82.696, 139.62, 81.305, 7.327]
  Call Extruder(399.40175)
  MoveL 8514 to (-34.45, 161.76, 125.68) mm, rotated rx -180 ry 0 rz -180 deg; joints [-140.244, 71.348, -82.691, 139.687, 81.304, 7.31]
  MoveL 8515 to (-34.45, 161.76, 125.68) mm, rotated rx -180 ry 0 rz -180 deg; joints [-140.244, 71.348, -82.691, 139.687, 81.304, 7.31]
  Call Extruder(399.73518)
  MoveL 8516 to (-34.9, 161.43, 125.68) mm, rotated rx -180 ry 0 rz 180 deg; joints [-140.366, 71.357, -82.681, 139.812, 81.302, 7.28]
  MoveL 8517 to (-34.9, 161.43, 125.68) mm, rotated rx -180 ry 0 rz 180 deg; joints [-140.366, 71.357, -82.681, 139.812, 81.302, 7.28]
  Call Extruder(400.06980)
  MoveL 8518 to (-35.35, 161.1, 125.68) mm, rotated rx 180 ry 0 rz 180 deg; joints [-140.489, 71.366, -82.672, 139.936, 81.301, 7.249]
  Call Extruder(400.89771)
  MoveL 8519 to (-36.39, 160.19, 125.68) mm, rotated rx -180 ry 0 rz -180 deg; joints [-140.797, 71.38, -82.657, 140.249, 81.284, 7.183]
  Call Extruder(401.72565)
  MoveL 8520 to (-37.3, 159.15, 125.68) mm, rotated rx -180 ry 0 rz -180 deg; joints [-141.109, 71.384, -82.653, 140.562, 81.251, 7.131]
  Call Extruder(401.89295)
  MoveL 8521 to (-37.47, 158.93, 125.68) mm, rotated rx -180 ry 0 rz -180 deg; joints [-141.172, 71.383, -82.654, 140.626, 81.242, 7.123]
  MoveL 8522 to (-37.47, 158.93, 125.68) mm, rotated rx -180 ry 0 rz -180 deg; joints [-141.172, 71.383, -82.654, 140.626, 81.242, 7.123]
  Call Extruder(402.22638)
  MoveL 8523 to (-37.79, 158.48, 125.68) mm, rotated rx -180 ry 0 rz 180 deg; joints [-141.298, 71.381, -82.656, 140.752, 81.224, 7.106]
  MoveL 8524 to (-37.79, 158.48, 125.68) mm, rotated rx -180 ry 0 rz 180 deg; joints [-141.298, 71.381, -82.656, 140.752, 81.224, 7.106]
  Call Extruder(402.55863)
  MoveL 8525 to (-38.12, 158.03, 125.68) mm, rotated rx 180 ry 0 rz 180 deg; joints [-141.424, 71.38, -82.658, 140.878, 81.205, 7.088]
  MoveL 8526 to (-38.12, 158.03, 125.68) mm, rotated rx 180 ry 0 rz 180 deg; joints [-141.424, 71.38, -82.658, 140.878, 81.205, 7.088]
  Call Extruder(402.67630)
  MoveL 8527 to (-38.22, 157.85, 125.68) mm, rotated rx 180 ry 0 rz 180 deg; joints [-141.468, 71.378, -82.66, 140.922, 81.197, 7.084]
  MoveL 8528 to (-38.22, 157.85, 125.68) mm, rotated rx 180 ry 0 rz 180 deg; joints [-141.468, 71.378, -82.66, 140.922, 81.197, 7.084]
  Call Extruder(402.88403)
  MoveL 8529 to (-38.4, 157.55, 125.68) mm, rotated rx -180 ry 0 rz -180 deg; joints [-141.547, 71.375, -82.663, 141, 81.182, 7.076]
  MoveL 8530 to (-38.4, 157.55, 125.68) mm, rotated rx -180 ry 0 rz -180 deg; joints [-141.547, 71.375, -82.663, 141, 81.182, 7.076]
  Call Extruder(403.09097)
  MoveL 8531 to (-38.57, 157.25, 125.68) mm, rotated rx 180 ry 0 rz -180 deg; joints [-141.625, 71.371, -82.667, 141.079, 81.167, 7.068]
  MoveL 8532 to (-38.57, 157.25, 125.68) mm, rotated rx 180 ry 0 rz -180 deg; joints [-141.625, 71.371, -82.667, 141.079, 81.167, 7.068]
  Call Extruder(403.29714)
  MoveL 8533 to (-38.75, 156.94, 125.68) mm, rotated rx -180 ry 0 rz 180 deg; joints [-141.704, 71.368, -82.67, 141.157, 81.152, 7.061]
  MoveL 8534 to (-38.75, 156.94, 125.68) mm, rotated rx -180 ry 0 rz 180 deg; joints [-141.704, 71.368, -82.67, 141.157, 81.152, 7.061]
  Call Extruder(403.47882)
  MoveL 8535 to (-38.89, 156.66, 125.68) mm, rotated rx -180 ry 0 rz 180 deg; joints [-141.773, 71.364, -82.674, 141.225, 81.138, 7.055]
  MoveL 8536 to (-38.89, 156.66, 125.68) mm, rotated rx -180 ry 0 rz 180 deg; joints [-141.773, 71.364, -82.674, 141.225, 81.138, 7.055]
  Call Extruder(403.63681)
  MoveL 8537 to (-39, 156.42, 125.68) mm, rotated rx 180 ry 0 rz 180 deg; joints [-141.832, 71.36, -82.679, 141.284, 81.123, 7.052]
  MoveL 8538 to (-39, 156.42, 125.68) mm, rotated rx 180 ry 0 rz 180 deg; joints [-141.832, 71.36, -82.679, 141.284, 81.123, 7.052]
  Call Extruder(403.79419)
  MoveL 8539 to (-39.1, 156.17, 125.68) mm, rotated rx -180 ry 0 rz 180 deg; joints [-141.891, 71.355, -82.684, 141.343, 81.109, 7.048]
  MoveL 8540 to (-39.1, 156.17, 125.68) mm, rotated rx -180 ry 0 rz 180 deg; joints [-141.891, 71.355, -82.684, 141.343, 81.109, 7.048]
  Call Extruder(403.97691)
  MoveL 8541 to (-39.23, 155.87, 125.68) mm, rotated rx -180 ry 0 rz 180 deg; joints [-141.96, 71.35, -82.689, 141.411, 81.091, 7.045]
  MoveL 8542 to (-39.23, 155.87, 125.68) mm, rotated rx -180 ry 0 rz 180 deg; joints [-141.96, 71.35, -82.689, 141.411, 81.091, 7.045]
  Call Extruder(404.15887)
  MoveL 8543 to (-39.35, 155.58, 125.68) mm, rotated rx 180 ry 0 rz 180 deg; joints [-142.029, 71.344, -82.695, 141.479, 81.074, 7.041]
  MoveL 8544 to (-39.35, 155.58, 125.68) mm, rotated rx 180 ry 0 rz 180 deg; joints [-142.029, 71.344, -82.695, 141.479, 81.074, 7.041]
  Call Extruder(404.30621)
  MoveL 8545 to (-39.44, 155.34, 125.68) mm, rotated rx -180 ry 0 rz 180 deg; joints [-142.085, 71.34, -82.7, 141.534, 81.06, 7.038]
  MoveL 8546 to (-39.44, 155.34, 125.68) mm, rotated rx -180 ry 0 rz 180 deg; joints [-142.085, 71.34, -82.7, 141.534, 81.06, 7.038]
  Call Extruder(404.41944)
  MoveL 8547 to (-39.5, 155.15, 125.68) mm, rotated rx -180 ry 0 rz -180 deg; joints [-142.127, 71.335, -82.705, 141.576, 81.048, 7.037]
  MoveL 8548 to (-39.5, 155.15, 125.68) mm, rotated rx -180 ry 0 rz -180 deg; joints [-142.127, 71.335, -82.705, 141.576, 81.048, 7.037]
  Call Extruder(404.53223)
  MoveL 8549 to (-39.56, 154.97, 125.68) mm, rotated rx 180 ry 0 rz 180 deg; joints [-142.169, 71.331, -82.709, 141.617, 81.036, 7.036]
  MoveL 8550 to (-39.56, 154.97, 125.68) mm, rotated rx 180 ry 0 rz 180 deg; joints [-142.169, 71.331, -82.709, 141.617, 81.036, 7.036]
  Call Extruder(404.64458)
  MoveL 8551 to (-39.62, 154.78, 125.68) mm, rotated rx 180 ry 0 rz 180 deg; joints [-142.212, 71.327, -82.714, 141.659, 81.023, 7.035]
  MoveL 8552 to (-39.62, 154.78, 125.68) mm, rotated rx 180 ry 0 rz 180 deg; joints [-142.212, 71.327, -82.714, 141.659, 81.023, 7.035]
  Call Extruder(404.75648)
  MoveL 8553 to (-39.68, 154.59, 125.68) mm, rotated rx 180 ry 0 rz -180 deg; joints [-142.254, 71.322, -82.718, 141.7, 81.011, 7.034]
  MoveL 8554 to (-39.68, 154.59, 125.68) mm, rotated rx 180 ry 0 rz -180 deg; joints [-142.254, 71.322, -82.718, 141.7, 81.011, 7.034]
  Call Extruder(404.87788)
  MoveL 8555 to (-39.75, 154.38, 125.68) mm, rotated rx 180 ry 0 rz 180 deg; joints [-142.3, 71.318, -82.723, 141.745, 80.998, 7.033]
  MoveL 8556 to (-39.75, 154.38, 125.68) mm, rotated rx 180 ry 0 rz 180 deg; joints [-142.3, 71.318, -82.723, 141.745, 80.998, 7.033]
  Call Extruder(405.00867)
  MoveL 8557 to (-39.81, 154.16, 125.68) mm, rotated rx 180 ry 0 rz 180 deg; joints [-142.35, 71.312, -82.729, 141.794, 80.983, 7.032]
  MoveL 8558 to (-39.81, 154.16, 125.68) mm, rotated rx 180 ry 0 rz 180 deg; joints [-142.35, 71.312, -82.729, 141.794, 80.983, 7.032]
  Call Extruder(405.13890)
  MoveL 8559 to (-39.88, 153.94, 125.68) mm, rotated rx -180 ry 0 rz 180 deg; joints [-142.399, 71.307, -82.735, 141.843, 80.969, 7.031]
  MoveL 8560 to (-39.88, 153.94, 125.68) mm, rotated rx -180 ry 0 rz 180 deg; joints [-142.399, 71.307, -82.735, 141.843, 80.969, 7.031]
  Call Extruder(405.26856)
  MoveL 8561 to (-39.95, 153.71, 125.68) mm, rotated rx 180 ry 0 rz 180 deg; joints [-142.449, 71.302, -82.74, 141.892, 80.954, 7.03]
  MoveL 8562 to (-39.95, 153.71, 125.68) mm, rotated rx 180 ry 0 rz 180 deg; joints [-142.449, 71.302, -82.74, 141.892, 80.954, 7.03]
  Call Extruder(405.39766)
  MoveL 8563 to (-40.02, 153.49, 125.68) mm, rotated rx -180 ry 0 rz -180 deg; joints [-142.498, 71.296, -82.746, 141.941, 80.939, 7.029]
  MoveL 8564 to (-40.02, 153.49, 125.68) mm, rotated rx -180 ry 0 rz -180 deg; joints [-142.498, 71.296, -82.746, 141.941, 80.939, 7.029]
  Call Extruder(405.51275)
  MoveL 8565 to (-40.06, 153.28, 125.68) mm, rotated rx -180 ry 0 rz -180 deg; joints [-142.541, 71.291, -82.752, 141.983, 80.925, 7.029]
  MoveL 8566 to (-40.06, 153.28, 125.68) mm, rotated rx -180 ry 0 rz -180 deg; joints [-142.541, 71.291, -82.752, 141.983, 80.925, 7.029]
  Call Extruder(405.62739)
  MoveL 8567 to (-40.11, 153.08, 125.68) mm, rotated rx -180 ry 0 rz 180 deg; joints [-142.584, 71.285, -82.758, 142.025, 80.911, 7.03]
  MoveL 8568 to (-40.11, 153.08, 125.68) mm, rotated rx -180 ry 0 rz 180 deg; joints [-142.584, 71.285, -82.758, 142.025, 80.911, 7.03]
  Call Extruder(405.74157)
  MoveL 8569 to (-40.15, 152.88, 125.68) mm, rotated rx 180 ry 0 rz -180 deg; joints [-142.627, 71.279, -82.764, 142.067, 80.896, 7.03]
  MoveL 8570 to (-40.15, 152.88, 125.68) mm, rotated rx 180 ry 0 rz -180 deg; joints [-142.627, 71.279, -82.764, 142.067, 80.896, 7.03]
  Call Extruder(405.85530)
  MoveL 8571 to (-40.2, 152.67, 125.68) mm, rotated rx -180 ry 0 rz 180 deg; joints [-142.671, 71.274, -82.77, 142.109, 80.882, 7.031]
  MoveL 8572 to (-40.2, 152.67, 125.68) mm, rotated rx -180 ry 0 rz 180 deg; joints [-142.671, 71.274, -82.77, 142.109, 80.882, 7.031]
  Call Extruder(405.98072)
  MoveL 8573 to (-40.24, 152.45, 125.68) mm, rotated rx 180 ry 0 rz 180 deg; joints [-142.718, 71.267, -82.776, 142.156, 80.865, 7.031]
  MoveL 8574 to (-40.24, 152.45, 125.68) mm, rotated rx 180 ry 0 rz 180 deg; joints [-142.718, 71.267, -82.776, 142.156, 80.865, 7.031]
  Call Extruder(406.11770)
  MoveL 8575 to (-40.29, 152.2, 125.68) mm, rotated rx -180 ry 0 rz -180 deg; joints [-142.77, 71.26, -82.784, 142.206, 80.848, 7.032]
  MoveL 8576 to (-40.29, 152.2, 125.68) mm, rotated rx -180 ry 0 rz -180 deg; joints [-142.77, 71.26, -82.784, 142.206, 80.848, 7.032]
  Call Extruder(406.25406)
  MoveL 8577 to (-40.34, 151.95, 125.68) mm, rotated rx -180 ry 0 rz -180 deg; joints [-142.822, 71.253, -82.791, 142.257, 80.83, 7.033]
  MoveL 8578 to (-40.34, 151.95, 125.68) mm, rotated rx -180 ry 0 rz -180 deg; joints [-142.822, 71.253, -82.791, 142.257, 80.83, 7.033]
  Call Extruder(406.38982)
  MoveL 8579 to (-40.39, 151.7, 125.68) mm, rotated rx -180 ry 0 rz 180 deg; joints [-142.874, 71.246, -82.799, 142.308, 80.812, 7.033]
  MoveL 8580 to (-40.39, 151.7, 125.68) mm, rotated rx -180 ry 0 rz 180 deg; joints [-142.874, 71.246, -82.799, 142.308, 80.812, 7.033]
  Call Extruder(406.52496)
  MoveL 8581 to (-40.44, 151.45, 125.68) mm, rotated rx -180 ry 0 rz 180 deg; joints [-142.926, 71.239, -82.806, 142.359, 80.794, 7.034]
  MoveL 8582 to (-40.44, 151.45, 125.68) mm, rotated rx -180 ry 0 rz 180 deg; joints [-142.926, 71.239, -82.806, 142.359, 80.794, 7.034]
  Call Extruder(406.65950)
  MoveL 8583 to (-40.49, 151.2, 125.68) mm, rotated rx 180 ry 0 rz -180 deg; joints [-142.978, 71.232, -82.813, 142.41, 80.776, 7.035]
  MoveL 8584 to (-40.49, 151.2, 125.68) mm, rotated rx 180 ry 0 rz -180 deg; joints [-142.978, 71.232, -82.813, 142.41, 80.776, 7.035]
  Call Extruder(406.79342)
  MoveL 8585 to (-40.54, 150.95, 125.68) mm, rotated rx 180 ry 0 rz 180 deg; joints [-143.031, 71.224, -82.821, 142.461, 80.758, 7.035]
  MoveL 8586 to (-40.54, 150.95, 125.68) mm, rotated rx 180 ry 0 rz 180 deg; joints [-143.031, 71.224, -82.821, 142.461, 80.758, 7.035]
  Call Extruder(406.94128)
  MoveL 8587 to (-40.59, 150.67, 125.68) mm, rotated rx -180 ry 0 rz -180 deg; joints [-143.088, 71.216, -82.829, 142.517, 80.738, 7.036]
  MoveL 8588 to (-40.59, 150.67, 125.68) mm, rotated rx -180 ry 0 rz -180 deg; joints [-143.088, 71.216, -82.829, 142.517, 80.738, 7.036]
  Call Extruder(407.10301)
  MoveL 8589 to (-40.64, 150.37, 125.68) mm, rotated rx -180 ry 0 rz 180 deg; joints [-143.15, 71.207, -82.839, 142.578, 80.715, 7.038]
  MoveL 8590 to (-40.64, 150.37, 125.68) mm, rotated rx -180 ry 0 rz 180 deg; joints [-143.15, 71.207, -82.839, 142.578, 80.715, 7.038]
  Call Extruder(407.26400)
  MoveL 8591 to (-40.69, 150.06, 125.68) mm, rotated rx -180 ry 0 rz 180 deg; joints [-143.213, 71.198, -82.849, 142.639, 80.692, 7.039]
  MoveL 8592 to (-40.69, 150.06, 125.68) mm, rotated rx -180 ry 0 rz 180 deg; joints [-143.213, 71.198, -82.849, 142.639, 80.692, 7.039]
  Call Extruder(407.42427)
  MoveL 8593 to (-40.74, 149.76, 125.68) mm, rotated rx 180 ry 0 rz 180 deg; joints [-143.276, 71.188, -82.858, 142.7, 80.67, 7.041]
  MoveL 8594 to (-40.74, 149.76, 125.68) mm, rotated rx 180 ry 0 rz 180 deg; joints [-143.276, 71.188, -82.858, 142.7, 80.67, 7.041]
  Call Extruder(407.58382)
  MoveL 8595 to (-40.78, 149.45, 125.68) mm, rotated rx -180 ry 0 rz 180 deg; joints [-143.338, 71.179, -82.868, 142.762, 80.647, 7.042]
  MoveL 8596 to (-40.78, 149.45, 125.68) mm, rotated rx -180 ry 0 rz 180 deg; joints [-143.338, 71.179, -82.868, 142.762, 80.647, 7.042]
  Call Extruder(407.74263)
  MoveL 8597 to (-40.83, 149.14, 125.68) mm, rotated rx -180 ry 0 rz -180 deg; joints [-143.401, 71.17, -82.877, 142.823, 80.624, 7.043]
  MoveL 8598 to (-40.83, 149.14, 125.68) mm, rotated rx -180 ry 0 rz -180 deg; joints [-143.401, 71.17, -82.877, 142.823, 80.624, 7.043]
  Call Extruder(407.92129)
  MoveL 8599 to (-40.88, 148.8, 125.68) mm, rotated rx -180 ry 0 rz -180 deg; joints [-143.471, 71.159, -82.889, 142.891, 80.598, 7.045]
  MoveL 8600 to (-40.88, 148.8, 125.68) mm, rotated rx -180 ry 0 rz -180 deg; joints [-143.471, 71.159, -82.889, 142.891, 80.598, 7.045]
  Call Extruder(408.11974)
  MoveL 8601 to (-40.93, 148.41, 125.68) mm, rotated rx 180 ry 0 rz 180 deg; joints [-143.549, 71.146, -82.902, 142.967, 80.568, 7.048]
  MoveL 8602 to (-40.93, 148.41, 125.68) mm, rotated rx 180 ry 0 rz 180 deg; joints [-143.549, 71.146, -82.902, 142.967, 80.568, 7.048]
  Call Extruder(408.31731)
  MoveL 8603 to (-40.97, 148.02, 125.68) mm, rotated rx 180 ry 0 rz -180 deg; joints [-143.627, 71.134, -82.914, 143.043, 80.538, 7.051]
  MoveL 8604 to (-40.97, 148.02, 125.68) mm, rotated rx 180 ry 0 rz -180 deg; joints [-143.627, 71.134, -82.914, 143.043, 80.538, 7.051]
  Call Extruder(408.51402)
  MoveL 8605 to (-41.02, 147.63, 125.68) mm, rotated rx -180 ry 0 rz -180 deg; joints [-143.705, 71.121, -82.927, 143.119, 80.509, 7.053]
  MoveL 8606 to (-41.02, 147.63, 125.68) mm, rotated rx -180 ry 0 rz -180 deg; joints [-143.705, 71.121, -82.927, 143.119, 80.509, 7.053]
  Call Extruder(408.70985)
  MoveL 8607 to (-41.06, 147.25, 125.68) mm, rotated rx 180 ry 0 rz -180 deg; joints [-143.783, 71.109, -82.94, 143.194, 80.479, 7.056]
  MoveL 8608 to (-41.06, 147.25, 125.68) mm, rotated rx 180 ry 0 rz -180 deg; joints [-143.783, 71.109, -82.94, 143.194, 80.479, 7.056]
  Call Extruder(409.00525)
  MoveL 8609 to (-41.11, 146.66, 125.68) mm, rotated rx -180 ry 0 rz -180 deg; joints [-143.899, 71.089, -82.96, 143.307, 80.432, 7.061]
  MoveL 8610 to (-41.11, 146.66, 125.68) mm, rotated rx -180 ry 0 rz -180 deg; joints [-143.899, 71.089, -82.96, 143.307, 80.432, 7.061]
  Call Extruder(409.29932)
  MoveL 8611 to (-41.15, 146.07, 125.68) mm, rotated rx -180 ry 0 rz 180 deg; joints [-144.015, 71.068, -82.981, 143.42, 80.385, 7.066]
  MoveL 8612 to (-41.15, 146.07, 125.68) mm, rotated rx -180 ry 0 rz 180 deg; joints [-144.015, 71.068, -82.981, 143.42, 80.385, 7.066]
  Call Extruder(409.59205)
  MoveL 8613 to (-41.2, 145.48, 125.68) mm, rotated rx -180 ry 0 rz 180 deg; joints [-144.131, 71.048, -83.001, 143.533, 80.338, 7.071]
  MoveL 8614 to (-41.2, 145.48, 125.68) mm, rotated rx -180 ry 0 rz 180 deg; joints [-144.131, 71.048, -83.001, 143.533, 80.338, 7.071]
  Call Extruder(410.16551)
  MoveL 8615 to (-41.25, 144.32, 125.68) mm, rotated rx 180 ry 0 rz 180 deg; joints [-144.355, 71.006, -83.043, 143.75, 80.243, 7.083]
  MoveL 8616 to (-41.25, 144.32, 125.68) mm, rotated rx 180 ry 0 rz 180 deg; joints [-144.355, 71.006, -83.043, 143.75, 80.243, 7.083]
  Call Extruder(410.87946)
  MoveL 8617 to (-41.29, 142.86, 125.68) mm, rotated rx 180 ry 0 rz 180 deg; joints [-144.635, 70.953, -83.097, 144.021, 80.122, 7.099]
  Call Extruder(452.94428)
  MoveL 8618 to (-41.29, 57.14, 125.68) mm, rotated rx 180 ry 0 rz 180 deg; joints [-164.153, 68.244, -85.288, 163.464, 73.622, 4.786]
  Call Extruder(453.37284)
  MoveL 8619 to (-41.27, 56.26, 125.68) mm, rotated rx -180 ry 0 rz 180 deg; joints [-164.382, 68.224, -85.301, 163.699, 73.571, 4.728]
  MoveL 8620 to (-41.27, 56.26, 125.68) mm, rotated rx -180 ry 0 rz 180 deg; joints [-164.382, 68.224, -85.301, 163.699, 73.571, 4.728]
  Call Extruder(453.94629)
  MoveL 8621 to (-41.23, 55.1, 125.68) mm, rotated rx -180 ry 0 rz 180 deg; joints [-164.686, 68.196, -85.32, 164.011, 73.502, 4.652]
  MoveL 8622 to (-41.23, 55.1, 125.68) mm, rotated rx -180 ry 0 rz 180 deg; joints [-164.686, 68.196, -85.32, 164.011, 73.502, 4.652]
  Call Extruder(454.38061)
  MoveL 8623 to (-41.18, 54.23, 125.68) mm, rotated rx 180 ry 0 rz 180 deg; joints [-164.915, 68.175, -85.333, 164.246, 73.45, 4.594]
  MoveL 8624 to (-41.18, 54.23, 125.68) mm, rotated rx 180 ry 0 rz 180 deg; joints [-164.915, 68.175, -85.333, 164.246, 73.45, 4.594]
  Call Extruder(454.67467)
  MoveL 8625 to (-41.13, 53.64, 125.68) mm, rotated rx -180 ry 0 rz 180 deg; joints [-165.068, 68.159, -85.344, 164.404, 73.413, 4.556]
  MoveL 8626 to (-41.13, 53.64, 125.68) mm, rotated rx -180 ry 0 rz 180 deg; joints [-165.068, 68.159, -85.344, 164.404, 73.413, 4.556]
  Call Extruder(454.97007)
  MoveL 8627 to (-41.09, 53.05, 125.68) mm, rotated rx -180 ry 0 rz 180 deg; joints [-165.222, 68.144, -85.354, 164.562, 73.376, 4.517]
  MoveL 8628 to (-41.09, 53.05, 125.68) mm, rotated rx -180 ry 0 rz 180 deg; joints [-165.222, 68.144, -85.354, 164.562, 73.376, 4.517]
  Call Extruder(455.21630)
  MoveL 8629 to (-41.04, 52.56, 125.68) mm, rotated rx 180 ry 0 rz -180 deg; joints [-165.349, 68.13, -85.362, 164.692, 73.345, 4.486]
  MoveL 8630 to (-41.04, 52.56, 125.68) mm, rotated rx 180 ry 0 rz -180 deg; joints [-165.349, 68.13, -85.362, 164.692, 73.345, 4.486]
  Call Extruder(455.41301)
  MoveL 8631 to (-40.99, 52.17, 125.68) mm, rotated rx -180 ry 0 rz -180 deg; joints [-165.449, 68.119, -85.369, 164.795, 73.32, 4.461]
  MoveL 8632 to (-40.99, 52.17, 125.68) mm, rotated rx -180 ry 0 rz -180 deg; joints [-165.449, 68.119, -85.369, 164.795, 73.32, 4.461]
  Call Extruder(455.61058)
  MoveL 8633 to (-40.95, 51.78, 125.68) mm, rotated rx -180 ry 0 rz 180 deg; joints [-165.549, 68.108, -85.376, 164.898, 73.294, 4.436]
  MoveL 8634 to (-40.95, 51.78, 125.68) mm, rotated rx -180 ry 0 rz 180 deg; joints [-165.549, 68.108, -85.376, 164.898, 73.294, 4.436]
  Call Extruder(455.80903)
  MoveL 8635 to (-40.9, 51.4, 125.68) mm, rotated rx 180 ry 0 rz -180 deg; joints [-165.65, 68.097, -85.384, 165.001, 73.269, 4.411]
  MoveL 8636 to (-40.9, 51.4, 125.68) mm, rotated rx 180 ry 0 rz -180 deg; joints [-165.65, 68.097, -85.384, 165.001, 73.269, 4.411]
  Call Extruder(456.00833)
  MoveL 8637 to (-40.86, 51.01, 125.68) mm, rotated rx -180 ry 0 rz -180 deg; joints [-165.751, 68.086, -85.391, 165.104, 73.244, 4.385]
  MoveL 8638 to (-40.86, 51.01, 125.68) mm, rotated rx -180 ry 0 rz -180 deg; joints [-165.751, 68.086, -85.391, 165.104, 73.244, 4.385]
  Call Extruder(456.16715)
  MoveL 8639 to (-40.81, 50.7, 125.68) mm, rotated rx 180 ry 0 rz -180 deg; joints [-165.829, 68.076, -85.397, 165.185, 73.222, 4.366]
  MoveL 8640 to (-40.81, 50.7, 125.68) mm, rotated rx 180 ry 0 rz -180 deg; joints [-165.829, 68.076, -85.397, 165.185, 73.222, 4.366]
  Call Extruder(456.32669)
  MoveL 8641 to (-40.76, 50.4, 125.68) mm, rotated rx -180 ry 0 rz -180 deg; joints [-165.908, 68.067, -85.403, 165.266, 73.201, 4.346]
  MoveL 8642 to (-40.76, 50.4, 125.68) mm, rotated rx -180 ry 0 rz -180 deg; joints [-165.908, 68.067, -85.403, 165.266, 73.201, 4.346]
  Call Extruder(456.48696)
  MoveL 8643 to (-40.71, 50.09, 125.68) mm, rotated rx 180 ry 0 rz 180 deg; joints [-165.987, 68.057, -85.409, 165.347, 73.18, 4.327]
  MoveL 8644 to (-40.71, 50.09, 125.68) mm, rotated rx 180 ry 0 rz 180 deg; joints [-165.987, 68.057, -85.409, 165.347, 73.18, 4.327]
  Call Extruder(456.64796)
  MoveL 8645 to (-40.66, 49.79, 125.68) mm, rotated rx -180 ry 0 rz -180 deg; joints [-166.066, 68.048, -85.415, 165.428, 73.159, 4.307]
  MoveL 8646 to (-40.66, 49.79, 125.68) mm, rotated rx -180 ry 0 rz -180 deg; joints [-166.066, 68.048, -85.415, 165.428, 73.159, 4.307]
  Call Extruder(456.80968)
  MoveL 8647 to (-40.61, 49.48, 125.68) mm, rotated rx -180 ry 0 rz 180 deg; joints [-166.145, 68.038, -85.421, 165.509, 73.138, 4.287]
  MoveL 8648 to (-40.61, 49.48, 125.68) mm, rotated rx -180 ry 0 rz 180 deg; joints [-166.145, 68.038, -85.421, 165.509, 73.138, 4.287]
  Call Extruder(456.97214)
  MoveL 8649 to (-40.57, 49.17, 125.68) mm, rotated rx -180 ry 0 rz -180 deg; joints [-166.224, 68.029, -85.427, 165.59, 73.117, 4.267]
  MoveL 8650 to (-40.57, 49.17, 125.68) mm, rotated rx -180 ry 0 rz -180 deg; joints [-166.224, 68.029, -85.427, 165.59, 73.117, 4.267]
  Call Extruder(457.10606)
  MoveL 8651 to (-40.52, 48.93, 125.68) mm, rotated rx 180 ry 0 rz 180 deg; joints [-166.288, 68.02, -85.433, 165.656, 73.099, 4.252]
  MoveL 8652 to (-40.52, 48.93, 125.68) mm, rotated rx 180 ry 0 rz 180 deg; joints [-166.288, 68.02, -85.433, 165.656, 73.099, 4.252]
  Call Extruder(457.24060)
  MoveL 8653 to (-40.47, 48.68, 125.68) mm, rotated rx -180 ry 0 rz -180 deg; joints [-166.352, 68.012, -85.438, 165.722, 73.081, 4.236]
  MoveL 8654 to (-40.47, 48.68, 125.68) mm, rotated rx -180 ry 0 rz -180 deg; joints [-166.352, 68.012, -85.438, 165.722, 73.081, 4.236]
  Call Extruder(457.37574)
  MoveL 8655 to (-40.42, 48.43, 125.68) mm, rotated rx -180 ry 0 rz -180 deg; joints [-166.416, 68.003, -85.443, 165.787, 73.063, 4.22]
  MoveL 8656 to (-40.42, 48.43, 125.68) mm, rotated rx -180 ry 0 rz -180 deg; joints [-166.416, 68.003, -85.443, 165.787, 73.063, 4.22]
  Call Extruder(457.51150)
  MoveL 8657 to (-40.37, 48.18, 125.68) mm, rotated rx -180 ry 0 rz 180 deg; joints [-166.48, 67.995, -85.449, 165.853, 73.045, 4.204]
  MoveL 8658 to (-40.37, 48.18, 125.68) mm, rotated rx -180 ry 0 rz 180 deg; joints [-166.48, 67.995, -85.449, 165.853, 73.045, 4.204]
  Call Extruder(457.64786)
  MoveL 8659 to (-40.32, 47.93, 125.68) mm, rotated rx 180 ry 0 rz 180 deg; joints [-166.544, 67.986, -85.454, 165.919, 73.027, 4.188]
  MoveL 8660 to (-40.32, 47.93, 125.68) mm, rotated rx 180 ry 0 rz 180 deg; joints [-166.544, 67.986, -85.454, 165.919, 73.027, 4.188]
  Call Extruder(457.78484)
  MoveL 8661 to (-40.27, 47.68, 125.68) mm, rotated rx 180 ry 0 rz -180 deg; joints [-166.608, 67.978, -85.459, 165.985, 73.009, 4.172]
  MoveL 8662 to (-40.27, 47.68, 125.68) mm, rotated rx 180 ry 0 rz -180 deg; joints [-166.608, 67.978, -85.459, 165.985, 73.009, 4.172]
  Call Extruder(457.92243)
  MoveL 8663 to (-40.22, 47.43, 125.68) mm, rotated rx -180 ry 0 rz 180 deg; joints [-166.673, 67.97, -85.465, 166.051, 72.991, 4.156]
  MoveL 8664 to (-40.22, 47.43, 125.68) mm, rotated rx -180 ry 0 rz 180 deg; joints [-166.673, 67.97, -85.465, 166.051, 72.991, 4.156]
  Call Extruder(458.03615)
  MoveL 8665 to (-40.17, 47.23, 125.68) mm, rotated rx -180 ry 0 rz -180 deg; joints [-166.725, 67.962, -85.469, 166.105, 72.976, 4.143]
  MoveL 8666 to (-40.17, 47.23, 125.68) mm, rotated rx -180 ry 0 rz -180 deg; joints [-166.725, 67.962, -85.469, 166.105, 72.976, 4.143]
  Call Extruder(458.15034)
  MoveL 8667 to (-40.13, 47.02, 125.68) mm, rotated rx -180 ry 0 rz 180 deg; joints [-166.778, 67.955, -85.474, 166.159, 72.96, 4.13]
  MoveL 8668 to (-40.13, 47.02, 125.68) mm, rotated rx -180 ry 0 rz 180 deg; joints [-166.778, 67.955, -85.474, 166.159, 72.96, 4.13]
  Call Extruder(458.26497)
  MoveL 8669 to (-40.08, 46.82, 125.68) mm, rotated rx -180 ry 0 rz -180 deg; joints [-166.83, 67.948, -85.478, 166.213, 72.945, 4.116]
  MoveL 8670 to (-40.08, 46.82, 125.68) mm, rotated rx -180 ry 0 rz -180 deg; joints [-166.83, 67.948, -85.478, 166.213, 72.945, 4.116]
  Call Extruder(458.38006)
  MoveL 8671 to (-40.04, 46.61, 125.68) mm, rotated rx -180 ry 0 rz -180 deg; joints [-166.883, 67.941, -85.483, 166.267, 72.93, 4.103]
  MoveL 8672 to (-40.04, 46.61, 125.68) mm, rotated rx -180 ry 0 rz -180 deg; joints [-166.883, 67.941, -85.483, 166.267, 72.93, 4.103]
  Call Extruder(458.50230)
  MoveL 8673 to (-39.98, 46.4, 125.68) mm, rotated rx 180 ry 0 rz 180 deg; joints [-166.937, 67.933, -85.488, 166.323, 72.913, 4.09]
  MoveL 8674 to (-39.98, 46.4, 125.68) mm, rotated rx 180 ry 0 rz 180 deg; joints [-166.937, 67.933, -85.488, 166.323, 72.913, 4.09]
  Call Extruder(458.63196)
  MoveL 8675 to (-39.92, 46.18, 125.68) mm, rotated rx -180 ry 0 rz -180 deg; joints [-166.994, 67.923, -85.494, 166.381, 72.895, 4.076]
  MoveL 8676 to (-39.92, 46.18, 125.68) mm, rotated rx -180 ry 0 rz -180 deg; joints [-166.994, 67.923, -85.494, 166.381, 72.895, 4.076]
  Call Extruder(458.76219)
  MoveL 8677 to (-39.85, 45.95, 125.68) mm, rotated rx 180 ry 0 rz -180 deg; joints [-167.051, 67.914, -85.499, 166.439, 72.876, 4.062]
  MoveL 8678 to (-39.85, 45.95, 125.68) mm, rotated rx 180 ry 0 rz -180 deg; joints [-167.051, 67.914, -85.499, 166.439, 72.876, 4.062]
  Call Extruder(458.89299)
  MoveL 8679 to (-39.78, 45.73, 125.68) mm, rotated rx -180 ry 0 rz -180 deg; joints [-167.107, 67.905, -85.505, 166.497, 72.858, 4.049]
  MoveL 8680 to (-39.78, 45.73, 125.68) mm, rotated rx -180 ry 0 rz -180 deg; joints [-167.107, 67.905, -85.505, 166.497, 72.858, 4.049]
  Call Extruder(459.02435)
  MoveL 8681 to (-39.71, 45.5, 125.68) mm, rotated rx -180 ry 0 rz 180 deg; joints [-167.164, 67.896, -85.511, 166.555, 72.839, 4.035]
  MoveL 8682 to (-39.71, 45.5, 125.68) mm, rotated rx -180 ry 0 rz 180 deg; joints [-167.164, 67.896, -85.511, 166.555, 72.839, 4.035]
  Call Extruder(459.13625)
  MoveL 8683 to (-39.65, 45.32, 125.68) mm, rotated rx -180 ry 0 rz -180 deg; joints [-167.212, 67.888, -85.516, 166.604, 72.823, 4.023]
  MoveL 8684 to (-39.65, 45.32, 125.68) mm, rotated rx -180 ry 0 rz -180 deg; joints [-167.212, 67.888, -85.516, 166.604, 72.823, 4.023]
  Call Extruder(459.24859)
  MoveL 8685 to (-39.59, 45.13, 125.68) mm, rotated rx -180 ry 0 rz 180 deg; joints [-167.26, 67.88, -85.521, 166.653, 72.807, 4.012]
  MoveL 8686 to (-39.59, 45.13, 125.68) mm, rotated rx -180 ry 0 rz 180 deg; joints [-167.26, 67.88, -85.521, 166.653, 72.807, 4.012]
  Call Extruder(459.36138)
  MoveL 8687 to (-39.53, 44.94, 125.68) mm, rotated rx -180 ry 0 rz -180 deg; joints [-167.307, 67.872, -85.526, 166.702, 72.791, 4]
  MoveL 8688 to (-39.53, 44.94, 125.68) mm, rotated rx -180 ry 0 rz -180 deg; joints [-167.307, 67.872, -85.526, 166.702, 72.791, 4]
  Call Extruder(459.47461)
  MoveL 8689 to (-39.47, 44.75, 125.68) mm, rotated rx -180 ry 0 rz 180 deg; joints [-167.355, 67.863, -85.531, 166.751, 72.775, 3.989]
  MoveL 8690 to (-39.47, 44.75, 125.68) mm, rotated rx -180 ry 0 rz 180 deg; joints [-167.355, 67.863, -85.531, 166.751, 72.775, 3.989]
  Call Extruder(459.58829)
  MoveL 8691 to (-39.41, 44.56, 125.68) mm, rotated rx -180 ry 0 rz 180 deg; joints [-167.403, 67.855, -85.536, 166.8, 72.759, 3.977]
  MoveL 8692 to (-39.41, 44.56, 125.68) mm, rotated rx -180 ry 0 rz 180 deg; joints [-167.403, 67.855, -85.536, 166.8, 72.759, 3.977]
  Call Extruder(459.77026)
  MoveL 8693 to (-39.29, 44.27, 125.68) mm, rotated rx -180 ry 0 rz 180 deg; joints [-167.475, 67.841, -85.545, 166.874, 72.731, 3.96]
  MoveL 8694 to (-39.29, 44.27, 125.68) mm, rotated rx -180 ry 0 rz 180 deg; joints [-167.475, 67.841, -85.545, 166.874, 72.731, 3.96]
  Call Extruder(459.95298)
  MoveL 8695 to (-39.17, 43.98, 125.68) mm, rotated rx -180 ry 0 rz -180 deg; joints [-167.548, 67.826, -85.554, 166.948, 72.703, 3.943]
  MoveL 8696 to (-39.17, 43.98, 125.68) mm, rotated rx -180 ry 0 rz -180 deg; joints [-167.548, 67.826, -85.554, 166.948, 72.703, 3.943]
  Call Extruder(460.12339)
  MoveL 8697 to (-39.05, 43.71, 125.68) mm, rotated rx -180 ry 0 rz -180 deg; joints [-167.615, 67.813, -85.562, 167.017, 72.677, 3.927]
  MoveL 8698 to (-39.05, 43.71, 125.68) mm, rotated rx -180 ry 0 rz -180 deg; joints [-167.615, 67.813, -85.562, 167.017, 72.677, 3.927]
  Call Extruder(460.28137)
  MoveL 8699 to (-38.94, 43.46, 125.68) mm, rotated rx -180 ry 0 rz -180 deg; joints [-167.677, 67.8, -85.57, 167.08, 72.653, 3.913]
  MoveL 8700 to (-38.94, 43.46, 125.68) mm, rotated rx -180 ry 0 rz -180 deg; joints [-167.677, 67.8, -85.57, 167.08, 72.653, 3.913]
  Call Extruder(460.43996)
  MoveL 8701 to (-38.84, 43.21, 125.68) mm, rotated rx 180 ry 0 rz -180 deg; joints [-167.739, 67.788, -85.578, 167.144, 72.629, 3.898]
  MoveL 8702 to (-38.84, 43.21, 125.68) mm, rotated rx 180 ry 0 rz -180 deg; joints [-167.739, 67.788, -85.578, 167.144, 72.629, 3.898]
  Call Extruder(460.64612)
  MoveL 8703 to (-38.66, 42.91, 125.68) mm, rotated rx 180 ry 0 rz -180 deg; joints [-167.813, 67.769, -85.589, 167.218, 72.594, 3.882]
  MoveL 8704 to (-38.66, 42.91, 125.68) mm, rotated rx 180 ry 0 rz -180 deg; joints [-167.813, 67.769, -85.589, 167.218, 72.594, 3.882]
  Call Extruder(460.85306)
  MoveL 8705 to (-38.49, 42.6, 125.68) mm, rotated rx 180 ry 0 rz 180 deg; joints [-167.886, 67.75, -85.601, 167.293, 72.56, 3.866]
  MoveL 8706 to (-38.49, 42.6, 125.68) mm, rotated rx 180 ry 0 rz 180 deg; joints [-167.886, 67.75, -85.601, 167.293, 72.56, 3.866]
  Call Extruder(461.06079)
  MoveL 8707 to (-38.31, 42.3, 125.68) mm, rotated rx -180 ry 0 rz -180 deg; joints [-167.96, 67.731, -85.612, 167.368, 72.525, 3.85]
  MoveL 8708 to (-38.31, 42.3, 125.68) mm, rotated rx -180 ry 0 rz -180 deg; joints [-167.96, 67.731, -85.612, 167.368, 72.525, 3.85]
  Call Extruder(461.26929)
  MoveL 8709 to (-38.14, 41.99, 125.68) mm, rotated rx 180 ry 0 rz -180 deg; joints [-168.033, 67.712, -85.624, 167.443, 72.49, 3.834]
  MoveL 8710 to (-38.14, 41.99, 125.68) mm, rotated rx 180 ry 0 rz -180 deg; joints [-168.033, 67.712, -85.624, 167.443, 72.49, 3.834]
  Call Extruder(461.44884)
  MoveL 8711 to (-37.96, 41.75, 125.68) mm, rotated rx -180 ry 0 rz -180 deg; joints [-168.091, 67.694, -85.635, 167.501, 72.459, 3.822]
  MoveL 8712 to (-37.96, 41.75, 125.68) mm, rotated rx -180 ry 0 rz -180 deg; joints [-168.091, 67.694, -85.635, 167.501, 72.459, 3.822]
  Call Extruder(461.78228)
  MoveL 8713 to (-37.63, 41.3, 125.68) mm, rotated rx 180 ry 0 rz -180 deg; joints [-168.197, 67.661, -85.655, 167.608, 72.399, 3.801]
  MoveL 8714 to (-37.63, 41.3, 125.68) mm, rotated rx 180 ry 0 rz -180 deg; joints [-168.197, 67.661, -85.655, 167.608, 72.399, 3.801]
  Call Extruder(462.11690)
  MoveL 8715 to (-37.3, 40.85, 125.68) mm, rotated rx 180 ry 0 rz 180 deg; joints [-168.304, 67.628, -85.675, 167.717, 72.34, 3.779]
  Call Extruder(462.94483)
  MoveL 8716 to (-36.39, 39.81, 125.68) mm, rotated rx -180 ry 0 rz 180 deg; joints [-168.541, 67.539, -85.728, 167.956, 72.186, 3.735]
  Call Extruder(463.77274)
  MoveL 8717 to (-35.35, 38.9, 125.68) mm, rotated rx -180 ry 0 rz -180 deg; joints [-168.739, 67.441, -85.785, 168.153, 72.022, 3.704]
  Call Extruder(463.94004)
  MoveL 8718 to (-35.13, 38.73, 125.68) mm, rotated rx -180 ry 0 rz 180 deg; joints [-168.773, 67.421, -85.797, 168.186, 71.988, 3.701]
  MoveL 8719 to (-35.13, 38.73, 125.68) mm, rotated rx -180 ry 0 rz 180 deg; joints [-168.773, 67.421, -85.797, 168.186, 71.988, 3.701]
  Call Extruder(464.27347)
  MoveL 8720 to (-34.68, 38.4, 125.68) mm, rotated rx -180 ry 0 rz 180 deg; joints [-168.84, 67.38, -85.821, 168.253, 71.92, 3.693]
  MoveL 8721 to (-34.68, 38.4, 125.68) mm, rotated rx -180 ry 0 rz 180 deg; joints [-168.84, 67.38, -85.821, 168.253, 71.92, 3.693]
  Call Extruder(464.60571)
  MoveL 8722 to (-34.23, 38.08, 125.68) mm, rotated rx -180 ry 0 rz 180 deg; joints [-168.908, 67.338, -85.845, 168.32, 71.851, 3.684]
  MoveL 8723 to (-34.23, 38.08, 125.68) mm, rotated rx -180 ry 0 rz 180 deg; joints [-168.908, 67.338, -85.845, 168.32, 71.851, 3.684]
  Call Extruder(464.72342)
  MoveL 8724 to (-34.05, 37.98, 125.68) mm, rotated rx 180 ry 0 rz 180 deg; joints [-168.927, 67.323, -85.853, 168.338, 71.827, 3.683]
  MoveL 8725 to (-34.05, 37.98, 125.68) mm, rotated rx 180 ry 0 rz 180 deg; joints [-168.927, 67.323, -85.853, 168.338, 71.827, 3.683]
  Call Extruder(464.93114)
  MoveL 8726 to (-33.75, 37.8, 125.68) mm, rotated rx -180 ry 0 rz 180 deg; joints [-168.96, 67.296, -85.869, 168.37, 71.783, 3.682]
  MoveL 8727 to (-33.75, 37.8, 125.68) mm, rotated rx -180 ry 0 rz 180 deg; joints [-168.96, 67.296, -85.869, 168.37, 71.783, 3.682]
  Call Extruder(465.13808)
  MoveL 8728 to (-33.45, 37.63, 125.68) mm, rotated rx 180 ry 0 rz 180 deg; joints [-168.993, 67.268, -85.884, 168.402, 71.739, 3.68]
  MoveL 8729 to (-33.45, 37.63, 125.68) mm, rotated rx 180 ry 0 rz 180 deg; joints [-168.993, 67.268, -85.884, 168.402, 71.739, 3.68]
  Call Extruder(465.34424)
  MoveL 8730 to (-33.14, 37.45, 125.68) mm, rotated rx 180 ry 0 rz -180 deg; joints [-169.026, 67.241, -85.9, 168.434, 71.695, 3.678]
  MoveL 8731 to (-33.14, 37.45, 125.68) mm, rotated rx 180 ry 0 rz -180 deg; joints [-169.026, 67.241, -85.9, 168.434, 71.695, 3.678]
  Call Extruder(465.52591)
  MoveL 8732 to (-32.87, 37.31, 125.68) mm, rotated rx -180 ry 0 rz -180 deg; joints [-169.052, 67.217, -85.914, 168.458, 71.655, 3.678]
  MoveL 8733 to (-32.87, 37.31, 125.68) mm, rotated rx -180 ry 0 rz -180 deg; joints [-169.052, 67.217, -85.914, 168.458, 71.655, 3.678]
  Call Extruder(465.68390)
  MoveL 8734 to (-32.62, 37.2, 125.68) mm, rotated rx 180 ry 0 rz 180 deg; joints [-169.068, 67.195, -85.926, 168.473, 71.621, 3.679]
  MoveL 8735 to (-32.62, 37.2, 125.68) mm, rotated rx 180 ry 0 rz 180 deg; joints [-169.068, 67.195, -85.926, 168.473, 71.621, 3.679]
  Call Extruder(465.84129)
  MoveL 8736 to (-32.37, 37.09, 125.68) mm, rotated rx 180 ry 0 rz 180 deg; joints [-169.085, 67.173, -85.938, 168.489, 71.586, 3.681]
  MoveL 8737 to (-32.37, 37.09, 125.68) mm, rotated rx 180 ry 0 rz 180 deg; joints [-169.085, 67.173, -85.938, 168.489, 71.586, 3.681]
  Call Extruder(465.98171)
  MoveL 8738 to (-32.14, 37, 125.68) mm, rotated rx -180 ry 0 rz 180 deg; joints [-169.099, 67.153, -85.949, 168.501, 71.555, 3.683]
